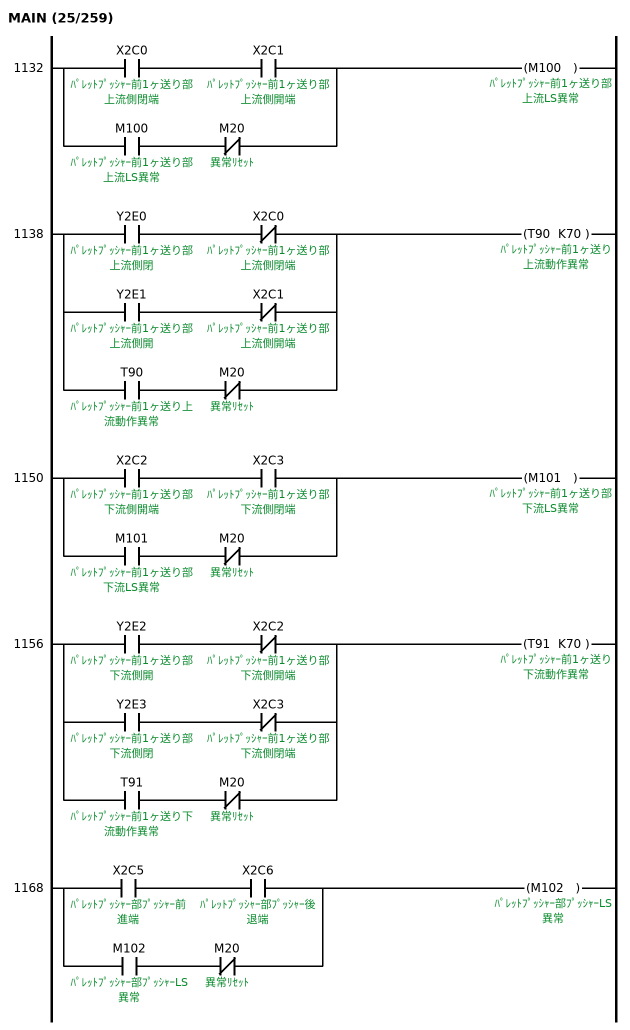
[picture p24: ladder of MAIN, rungs at steps 1132 to 1168]
1132  LD      X2C0  ; ﾊﾟﾚｯﾄﾌﾟｯｼｬｰ前1ヶ送り部上流側閉端
      AND     X2C1  ; ﾊﾟﾚｯﾄﾌﾟｯｼｬｰ前1ヶ送り部上流側開端
      LD      M100  ; ﾊﾟﾚｯﾄﾌﾟｯｼｬｰ前1ヶ送り部上流LS異常
      ANI     M20  ; 異常ﾘｾｯﾄ
      ORB
      OUT     M100  ; ﾊﾟﾚｯﾄﾌﾟｯｼｬｰ前1ヶ送り部上流LS異常
1138  LD      Y2E0  ; ﾊﾟﾚｯﾄﾌﾟｯｼｬｰ前1ヶ送り部上流側閉
      ANI     X2C0  ; ﾊﾟﾚｯﾄﾌﾟｯｼｬｰ前1ヶ送り部上流側閉端
      LD      Y2E1  ; ﾊﾟﾚｯﾄﾌﾟｯｼｬｰ前1ヶ送り部上流側開
      ANI     X2C1  ; ﾊﾟﾚｯﾄﾌﾟｯｼｬｰ前1ヶ送り部上流側開端
      ORB
      LD      T90  ; ﾊﾟﾚｯﾄﾌﾟｯｼｬｰ前1ヶ送り上流動作異常
      ANI     M20  ; 異常ﾘｾｯﾄ
      ORB
      OUT     T90 K70  ; ﾊﾟﾚｯﾄﾌﾟｯｼｬｰ前1ヶ送り上流動作異常
1150  LD      X2C2  ; ﾊﾟﾚｯﾄﾌﾟｯｼｬｰ前1ヶ送り部下流側開端
      AND     X2C3  ; ﾊﾟﾚｯﾄﾌﾟｯｼｬｰ前1ヶ送り部下流側閉端
      LD      M101  ; ﾊﾟﾚｯﾄﾌﾟｯｼｬｰ前1ヶ送り部下流LS異常
      ANI     M20  ; 異常ﾘｾｯﾄ
      ORB
      OUT     M101  ; ﾊﾟﾚｯﾄﾌﾟｯｼｬｰ前1ヶ送り部下流LS異常
1156  LD      Y2E2  ; ﾊﾟﾚｯﾄﾌﾟｯｼｬｰ前1ヶ送り部下流側開
      ANI     X2C2  ; ﾊﾟﾚｯﾄﾌﾟｯｼｬｰ前1ヶ送り部下流側開端
      LD      Y2E3  ; ﾊﾟﾚｯﾄﾌﾟｯｼｬｰ前1ヶ送り部下流側閉
      ANI     X2C3  ; ﾊﾟﾚｯﾄﾌﾟｯｼｬｰ前1ヶ送り部下流側閉端
      ORB
      LD      T91  ; ﾊﾟﾚｯﾄﾌﾟｯｼｬｰ前1ヶ送り下流動作異常
      ANI     M20  ; 異常ﾘｾｯﾄ
      ORB
      OUT     T91 K70  ; ﾊﾟﾚｯﾄﾌﾟｯｼｬｰ前1ヶ送り下流動作異常
1168  LD      X2C5  ; ﾊﾟﾚｯﾄﾌﾟｯｼｬｰ部ﾌﾟｯｼｬｰ前進端
      AND     X2C6  ; ﾊﾟﾚｯﾄﾌﾟｯｼｬｰ部ﾌﾟｯｼｬｰ後退端
      LD      M102  ; ﾊﾟﾚｯﾄﾌﾟｯｼｬｰ部ﾌﾟｯｼｬｰLS異常
      ANI     M20  ; 異常ﾘｾｯﾄ
      ORB
      OUT     M102  ; ﾊﾟﾚｯﾄﾌﾟｯｼｬｰ部ﾌﾟｯｼｬｰLS異常
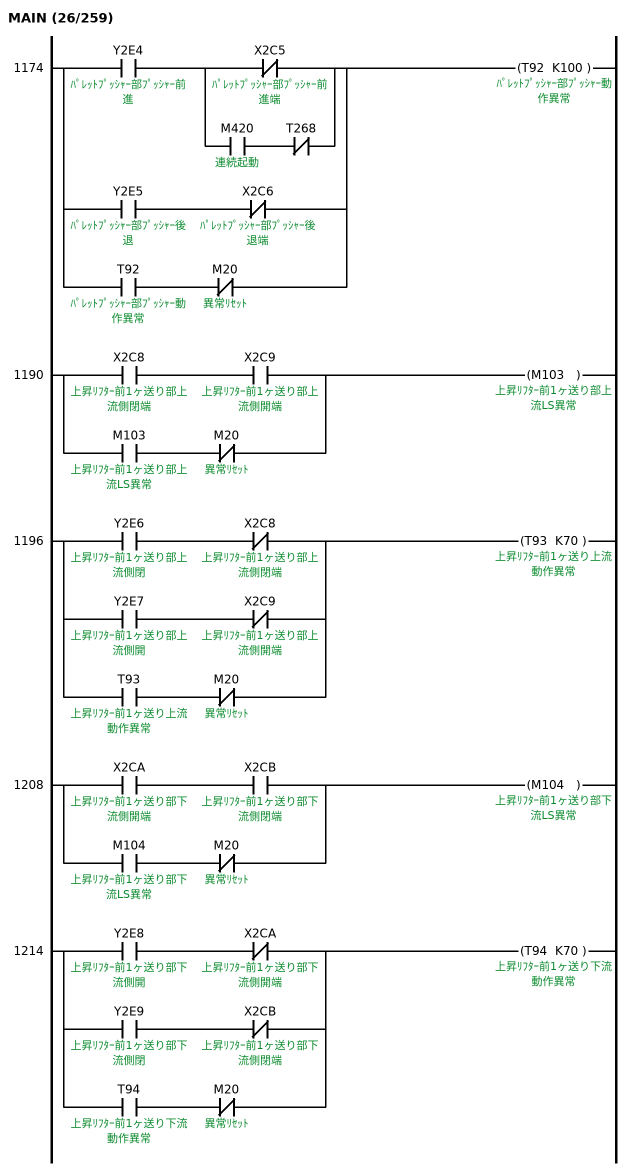
1174  LD      Y2E4  ; ﾊﾟﾚｯﾄﾌﾟｯｼｬｰ部ﾌﾟｯｼｬｰ前進
      LDI     X2C5  ; ﾊﾟﾚｯﾄﾌﾟｯｼｬｰ部ﾌﾟｯｼｬｰ前進端
      LD      M420  ; 連続起動
      ANI     T268
      ORB
      ANB
      LD      Y2E5  ; ﾊﾟﾚｯﾄﾌﾟｯｼｬｰ部ﾌﾟｯｼｬｰ後退
      ANI     X2C6  ; ﾊﾟﾚｯﾄﾌﾟｯｼｬｰ部ﾌﾟｯｼｬｰ後退端
      ORB
      LD      T92  ; ﾊﾟﾚｯﾄﾌﾟｯｼｬｰ部ﾌﾟｯｼｬｰ動作異常
      ANI     M20  ; 異常ﾘｾｯﾄ
      ORB
      OUT     T92 K100  ; ﾊﾟﾚｯﾄﾌﾟｯｼｬｰ部ﾌﾟｯｼｬｰ動作異常
1190  LD      X2C8  ; 上昇ﾘﾌﾀｰ前1ヶ送り部上流側閉端
      AND     X2C9  ; 上昇ﾘﾌﾀｰ前1ヶ送り部上流側開端
      LD      M103  ; 上昇ﾘﾌﾀｰ前1ヶ送り部上流LS異常
      ANI     M20  ; 異常ﾘｾｯﾄ
      ORB
      OUT     M103  ; 上昇ﾘﾌﾀｰ前1ヶ送り部上流LS異常
1196  LD      Y2E6  ; 上昇ﾘﾌﾀｰ前1ヶ送り部上流側閉
      ANI     X2C8  ; 上昇ﾘﾌﾀｰ前1ヶ送り部上流側閉端
      LD      Y2E7  ; 上昇ﾘﾌﾀｰ前1ヶ送り部上流側開
      ANI     X2C9  ; 上昇ﾘﾌﾀｰ前1ヶ送り部上流側開端
      ORB
      LD      T93  ; 上昇ﾘﾌﾀｰ前1ヶ送り上流動作異常
      ANI     M20  ; 異常ﾘｾｯﾄ
      ORB
      OUT     T93 K70  ; 上昇ﾘﾌﾀｰ前1ヶ送り上流動作異常
1208  LD      X2CA  ; 上昇ﾘﾌﾀｰ前1ヶ送り部下流側開端
      AND     X2CB  ; 上昇ﾘﾌﾀｰ前1ヶ送り部下流側閉端
      LD      M104  ; 上昇ﾘﾌﾀｰ前1ヶ送り部下流LS異常
      ANI     M20  ; 異常ﾘｾｯﾄ
      ORB
      OUT     M104  ; 上昇ﾘﾌﾀｰ前1ヶ送り部下流LS異常
1214  LD      Y2E8  ; 上昇ﾘﾌﾀｰ前1ヶ送り部下流側開
      ANI     X2CA  ; 上昇ﾘﾌﾀｰ前1ヶ送り部下流側開端
      LD      Y2E9  ; 上昇ﾘﾌﾀｰ前1ヶ送り部下流側閉
      ANI     X2CB  ; 上昇ﾘﾌﾀｰ前1ヶ送り部下流側閉端
      ORB
      LD      T94  ; 上昇ﾘﾌﾀｰ前1ヶ送り下流動作異常
      ANI     M20  ; 異常ﾘｾｯﾄ
      ORB
      OUT     T94 K70  ; 上昇ﾘﾌﾀｰ前1ヶ送り下流動作異常
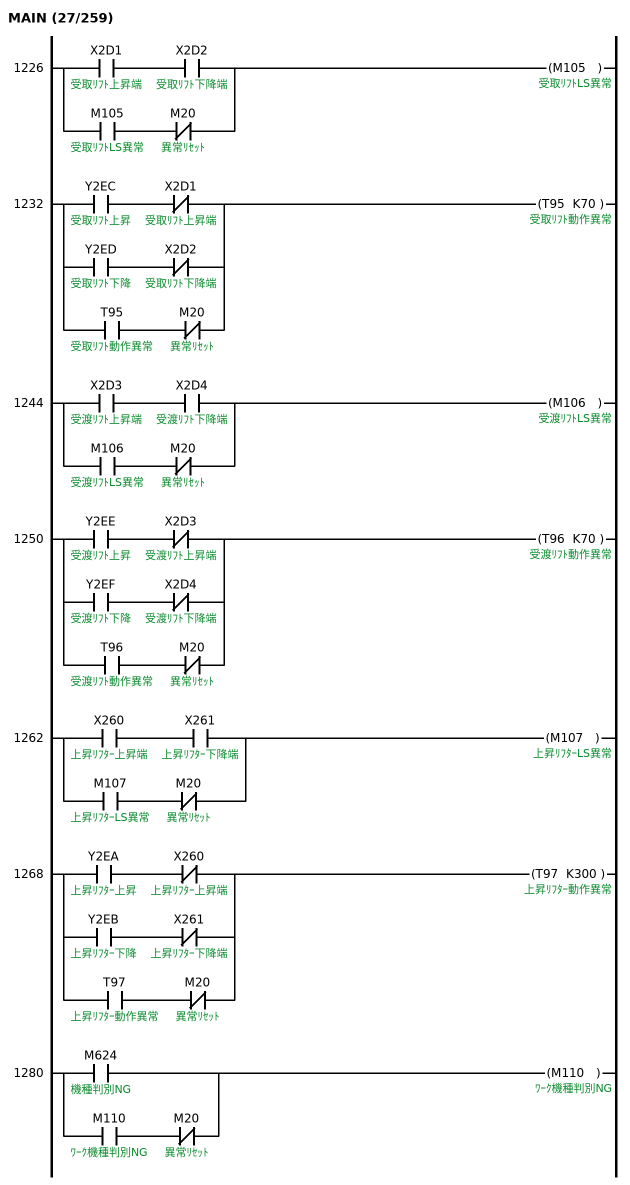
1226  LD      X2D1  ; 受取ﾘﾌﾄ上昇端
      AND     X2D2  ; 受取ﾘﾌﾄ下降端
      LD      M105  ; 受取ﾘﾌﾄLS異常
      ANI     M20  ; 異常ﾘｾｯﾄ
      ORB
      OUT     M105  ; 受取ﾘﾌﾄLS異常
1232  LD      Y2EC  ; 受取ﾘﾌﾄ上昇
      ANI     X2D1  ; 受取ﾘﾌﾄ上昇端
      LD      Y2ED  ; 受取ﾘﾌﾄ下降
      ANI     X2D2  ; 受取ﾘﾌﾄ下降端
      ORB
      LD      T95  ; 受取ﾘﾌﾄ動作異常
      ANI     M20  ; 異常ﾘｾｯﾄ
      ORB
      OUT     T95 K70  ; 受取ﾘﾌﾄ動作異常
1244  LD      X2D3  ; 受渡ﾘﾌﾄ上昇端
      AND     X2D4  ; 受渡ﾘﾌﾄ下降端
      LD      M106  ; 受渡ﾘﾌﾄLS異常
      ANI     M20  ; 異常ﾘｾｯﾄ
      ORB
      OUT     M106  ; 受渡ﾘﾌﾄLS異常
1250  LD      Y2EE  ; 受渡ﾘﾌﾄ上昇
      ANI     X2D3  ; 受渡ﾘﾌﾄ上昇端
      LD      Y2EF  ; 受渡ﾘﾌﾄ下降
      ANI     X2D4  ; 受渡ﾘﾌﾄ下降端
      ORB
      LD      T96  ; 受渡ﾘﾌﾄ動作異常
      ANI     M20  ; 異常ﾘｾｯﾄ
      ORB
      OUT     T96 K70  ; 受渡ﾘﾌﾄ動作異常
1262  LD      X260  ; 上昇ﾘﾌﾀｰ上昇端
      AND     X261  ; 上昇ﾘﾌﾀｰ下降端
      LD      M107  ; 上昇ﾘﾌﾀｰLS異常
      ANI     M20  ; 異常ﾘｾｯﾄ
      ORB
      OUT     M107  ; 上昇ﾘﾌﾀｰLS異常
1268  LD      Y2EA  ; 上昇ﾘﾌﾀｰ上昇
      ANI     X260  ; 上昇ﾘﾌﾀｰ上昇端
      LD      Y2EB  ; 上昇ﾘﾌﾀｰ下降
      ANI     X261  ; 上昇ﾘﾌﾀｰ下降端
      ORB
      LD      T97  ; 上昇ﾘﾌﾀｰ動作異常
      ANI     M20  ; 異常ﾘｾｯﾄ
      ORB
      OUT     T97 K300  ; 上昇ﾘﾌﾀｰ動作異常
1280  LD      M624  ; 機種判別NG
      LD      M110  ; ﾜｰｸ機種判別NG
      ANI     M20  ; 異常ﾘｾｯﾄ
      ORB
      OUT     M110  ; ﾜｰｸ機種判別NG
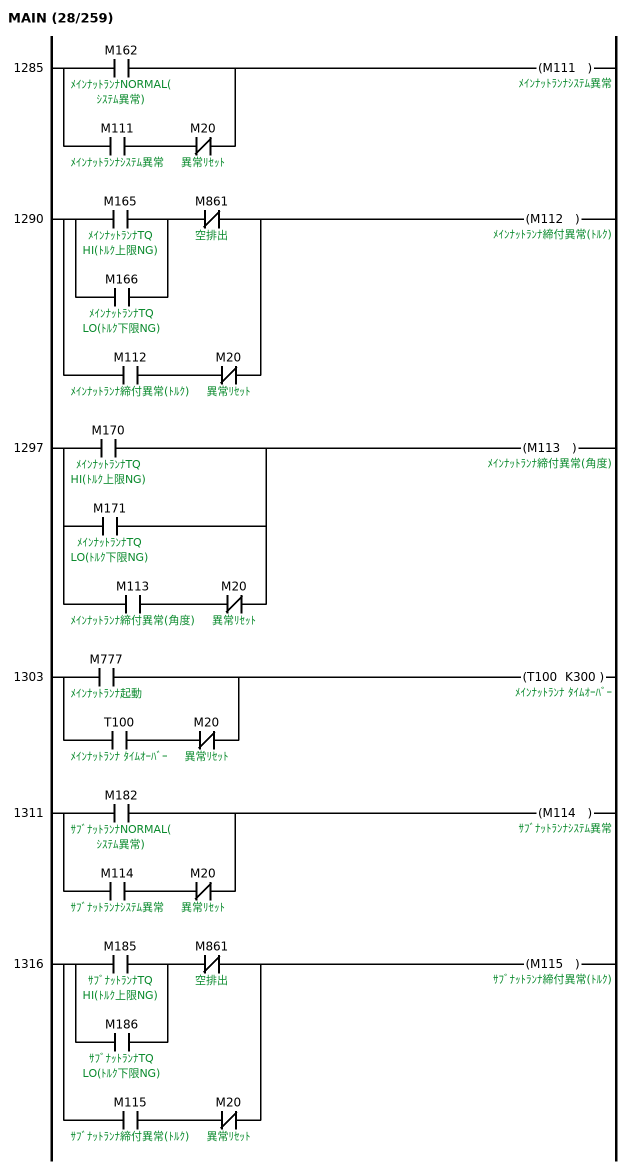
1285  LD      M162  ; ﾒｲﾝﾅｯﾄﾗﾝﾅNORMAL(ｼｽﾃﾑ異常)
      LD      M111  ; ﾒｲﾝﾅｯﾄﾗﾝﾅｼｽﾃﾑ異常
      ANI     M20  ; 異常ﾘｾｯﾄ
      ORB
      OUT     M111  ; ﾒｲﾝﾅｯﾄﾗﾝﾅｼｽﾃﾑ異常
1290  LD      M165  ; ﾒｲﾝﾅｯﾄﾗﾝﾅTQ HI(ﾄﾙｸ上限NG)
      OR      M166  ; ﾒｲﾝﾅｯﾄﾗﾝﾅTQ LO(ﾄﾙｸ下限NG)
      ANI     M861  ; 空排出
      LD      M112  ; ﾒｲﾝﾅｯﾄﾗﾝﾅ締付異常(ﾄﾙｸ)
      ANI     M20  ; 異常ﾘｾｯﾄ
      ORB
      OUT     M112  ; ﾒｲﾝﾅｯﾄﾗﾝﾅ締付異常(ﾄﾙｸ)
1297  LD      M170  ; ﾒｲﾝﾅｯﾄﾗﾝﾅTQ HI(ﾄﾙｸ上限NG)
      OR      M171  ; ﾒｲﾝﾅｯﾄﾗﾝﾅTQ LO(ﾄﾙｸ下限NG)
      LD      M113  ; ﾒｲﾝﾅｯﾄﾗﾝﾅ締付異常(角度)
      ANI     M20  ; 異常ﾘｾｯﾄ
      ORB
      OUT     M113  ; ﾒｲﾝﾅｯﾄﾗﾝﾅ締付異常(角度)
1303  LD      M777  ; ﾒｲﾝﾅｯﾄﾗﾝﾅ起動
      LD      T100  ; ﾒｲﾝﾅｯﾄﾗﾝﾅ ﾀｲﾑｵｰﾊﾞｰ
      ANI     M20  ; 異常ﾘｾｯﾄ
      ORB
      OUT     T100 K300  ; ﾒｲﾝﾅｯﾄﾗﾝﾅ ﾀｲﾑｵｰﾊﾞｰ
1311  LD      M182  ; ｻﾌﾞﾅｯﾄﾗﾝﾅNORMAL(ｼｽﾃﾑ異常)
      LD      M114  ; ｻﾌﾞﾅｯﾄﾗﾝﾅｼｽﾃﾑ異常
      ANI     M20  ; 異常ﾘｾｯﾄ
      ORB
      OUT     M114  ; ｻﾌﾞﾅｯﾄﾗﾝﾅｼｽﾃﾑ異常
1316  LD      M185  ; ｻﾌﾞﾅｯﾄﾗﾝﾅTQ HI(ﾄﾙｸ上限NG)
      OR      M186  ; ｻﾌﾞﾅｯﾄﾗﾝﾅTQ LO(ﾄﾙｸ下限NG)
      ANI     M861  ; 空排出
      LD      M115  ; ｻﾌﾞﾅｯﾄﾗﾝﾅ締付異常(ﾄﾙｸ)
      ANI     M20  ; 異常ﾘｾｯﾄ
      ORB
      OUT     M115  ; ｻﾌﾞﾅｯﾄﾗﾝﾅ締付異常(ﾄﾙｸ)
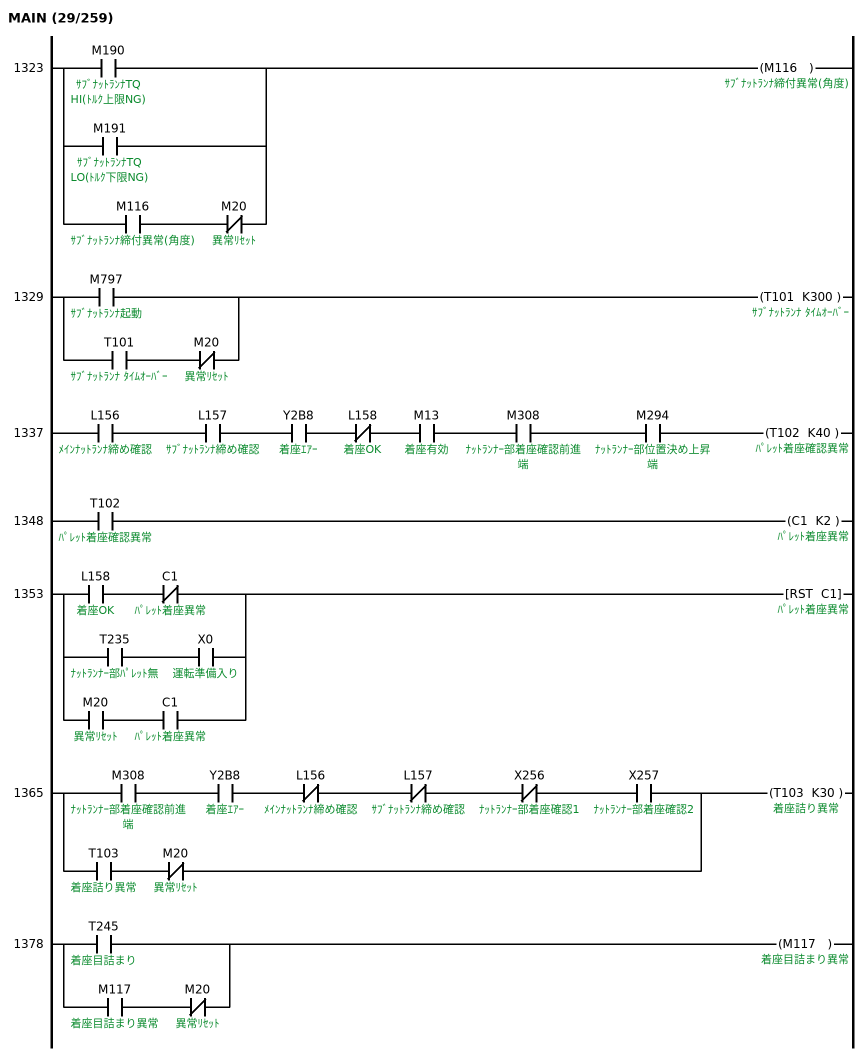
1323  LD      M190  ; ｻﾌﾞﾅｯﾄﾗﾝﾅTQ HI(ﾄﾙｸ上限NG)
      OR      M191  ; ｻﾌﾞﾅｯﾄﾗﾝﾅTQ LO(ﾄﾙｸ下限NG)
      LD      M116  ; ｻﾌﾞﾅｯﾄﾗﾝﾅ締付異常(角度)
      ANI     M20  ; 異常ﾘｾｯﾄ
      ORB
      OUT     M116  ; ｻﾌﾞﾅｯﾄﾗﾝﾅ締付異常(角度)
1329  LD      M797  ; ｻﾌﾞﾅｯﾄﾗﾝﾅ起動
      LD      T101  ; ｻﾌﾞﾅｯﾄﾗﾝﾅ ﾀｲﾑｵｰﾊﾞｰ
      ANI     M20  ; 異常ﾘｾｯﾄ
      ORB
      OUT     T101 K300  ; ｻﾌﾞﾅｯﾄﾗﾝﾅ ﾀｲﾑｵｰﾊﾞｰ
1337  LD      L156  ; ﾒｲﾝﾅｯﾄﾗﾝﾅ締め確認
      AND     L157  ; ｻﾌﾞﾅｯﾄﾗﾝﾅ締め確認
      AND     Y2B8  ; 着座ｴｱｰ
      ANI     L158  ; 着座OK
      AND     M13  ; 着座有効
      AND     M308  ; ﾅｯﾄﾗﾝﾅｰ部着座確認前進端
      AND     M294  ; ﾅｯﾄﾗﾝﾅｰ部位置決め上昇端
      OUT     T102 K40  ; ﾊﾟﾚｯﾄ着座確認異常
1348  LD      T102  ; ﾊﾟﾚｯﾄ着座確認異常
      OUT     C1 K2  ; ﾊﾟﾚｯﾄ着座異常
1353  LD      L158  ; 着座OK
      ANI     C1  ; ﾊﾟﾚｯﾄ着座異常
      LD      T235  ; ﾅｯﾄﾗﾝﾅｰ部ﾊﾟﾚｯﾄ無
      AND     X0  ; 運転準備入り
      ORB
      LD      M20  ; 異常ﾘｾｯﾄ
      AND     C1  ; ﾊﾟﾚｯﾄ着座異常
      ORB
      RST     C1  ; ﾊﾟﾚｯﾄ着座異常
1365  LD      M308  ; ﾅｯﾄﾗﾝﾅｰ部着座確認前進端
      AND     Y2B8  ; 着座ｴｱｰ
      ANI     L156  ; ﾒｲﾝﾅｯﾄﾗﾝﾅ締め確認
      ANI     L157  ; ｻﾌﾞﾅｯﾄﾗﾝﾅ締め確認
      ANI     X256  ; ﾅｯﾄﾗﾝﾅｰ部着座確認1
      AND     X257  ; ﾅｯﾄﾗﾝﾅｰ部着座確認2
      LD      T103  ; 着座詰り異常
      ANI     M20  ; 異常ﾘｾｯﾄ
      ORB
      OUT     T103 K30  ; 着座詰り異常
1378  LD      T245  ; 着座目詰まり
      LD      M117  ; 着座目詰まり異常
      ANI     M20  ; 異常ﾘｾｯﾄ
      ORB
      OUT     M117  ; 着座目詰まり異常
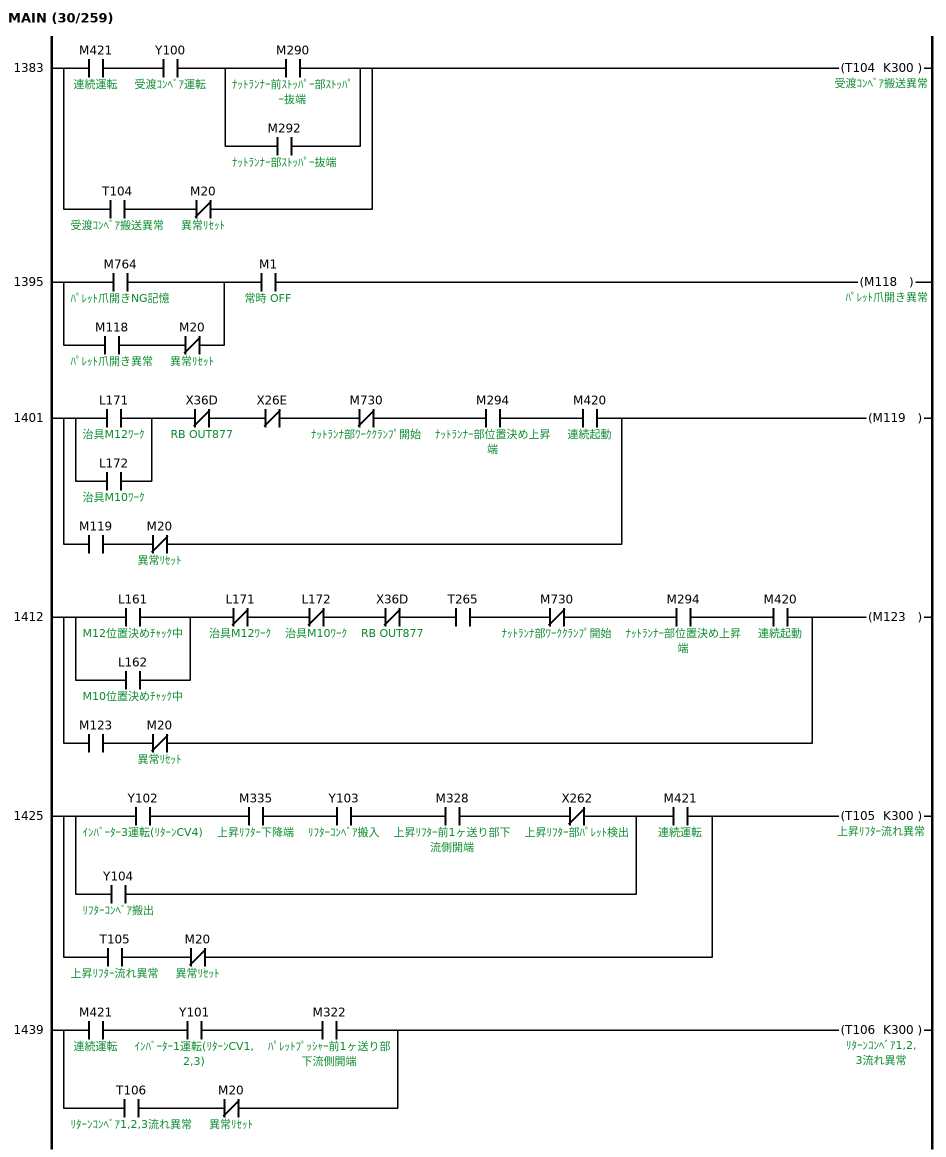
1383  LD      M421  ; 連続運転
      AND     Y100  ; 受渡ｺﾝﾍﾞｱ運転
      LD      M290  ; ﾅｯﾄﾗﾝﾅｰ前ｽﾄｯﾊﾟｰ部ｽﾄｯﾊﾟｰ抜端
      OR      M292  ; ﾅｯﾄﾗﾝﾅｰ部ｽﾄｯﾊﾟｰ抜端
      ANB
      LD      T104  ; 受渡ｺﾝﾍﾞｱ搬送異常
      ANI     M20  ; 異常ﾘｾｯﾄ
      ORB
      OUT     T104 K300  ; 受渡ｺﾝﾍﾞｱ搬送異常
1395  LD      M764  ; ﾊﾟﾚｯﾄ爪開きNG記憶
      LD      M118  ; ﾊﾟﾚｯﾄ爪開き異常
      ANI     M20  ; 異常ﾘｾｯﾄ
      ORB
      AND     M1  ; 常時 OFF
      OUT     M118  ; ﾊﾟﾚｯﾄ爪開き異常
1401  LD      L171  ; 治具M12ﾜｰｸ
      OR      L172  ; 治具M10ﾜｰｸ
      ANI     X36D  ; RB OUT877
      ANI     X26E
      ANI     M730  ; ﾅｯﾄﾗﾝﾅ部ﾜｰｸｸﾗﾝﾌﾟ開始
      AND     M294  ; ﾅｯﾄﾗﾝﾅｰ部位置決め上昇端
      AND     M420  ; 連続起動
      LD      M119
      ANI     M20  ; 異常ﾘｾｯﾄ
      ORB
      OUT     M119
1412  LD      L161  ; M12位置決めﾁｬｯｸ中
      OR      L162  ; M10位置決めﾁｬｯｸ中
      ANI     L171  ; 治具M12ﾜｰｸ
      ANI     L172  ; 治具M10ﾜｰｸ
      ANI     X36D  ; RB OUT877
      AND     T265
      ANI     M730  ; ﾅｯﾄﾗﾝﾅ部ﾜｰｸｸﾗﾝﾌﾟ開始
      AND     M294  ; ﾅｯﾄﾗﾝﾅｰ部位置決め上昇端
      AND     M420  ; 連続起動
      LD      M123
      ANI     M20  ; 異常ﾘｾｯﾄ
      ORB
      OUT     M123
1425  LD      Y102  ; ｲﾝﾊﾞｰﾀｰ3運転(ﾘﾀｰﾝCV4)
      AND     M335  ; 上昇ﾘﾌﾀｰ下降端
      AND     Y103  ; ﾘﾌﾀｰｺﾝﾍﾞｱ搬入
      AND     M328  ; 上昇ﾘﾌﾀｰ前1ヶ送り部下流側開端
      ANI     X262  ; 上昇ﾘﾌﾀｰ部ﾊﾟﾚｯﾄ検出
      OR      Y104  ; ﾘﾌﾀｰｺﾝﾍﾞｱ搬出
      AND     M421  ; 連続運転
      LD      T105  ; 上昇ﾘﾌﾀｰ流れ異常
      ANI     M20  ; 異常ﾘｾｯﾄ
      ORB
      OUT     T105 K300  ; 上昇ﾘﾌﾀｰ流れ異常
1439  LD      M421  ; 連続運転
      AND     Y101  ; ｲﾝﾊﾞｰﾀｰ1運転(ﾘﾀｰﾝCV1,2,3)
      AND     M322  ; ﾊﾟﾚｯﾄﾌﾟｯｼｬｰ前1ヶ送り部下流側開端
      LD      T106  ; ﾘﾀｰﾝｺﾝﾍﾞｱ1,2,3流れ異常
      ANI     M20  ; 異常ﾘｾｯﾄ
      ORB
      OUT     T106 K300  ; ﾘﾀｰﾝｺﾝﾍﾞｱ1,2,3流れ異常
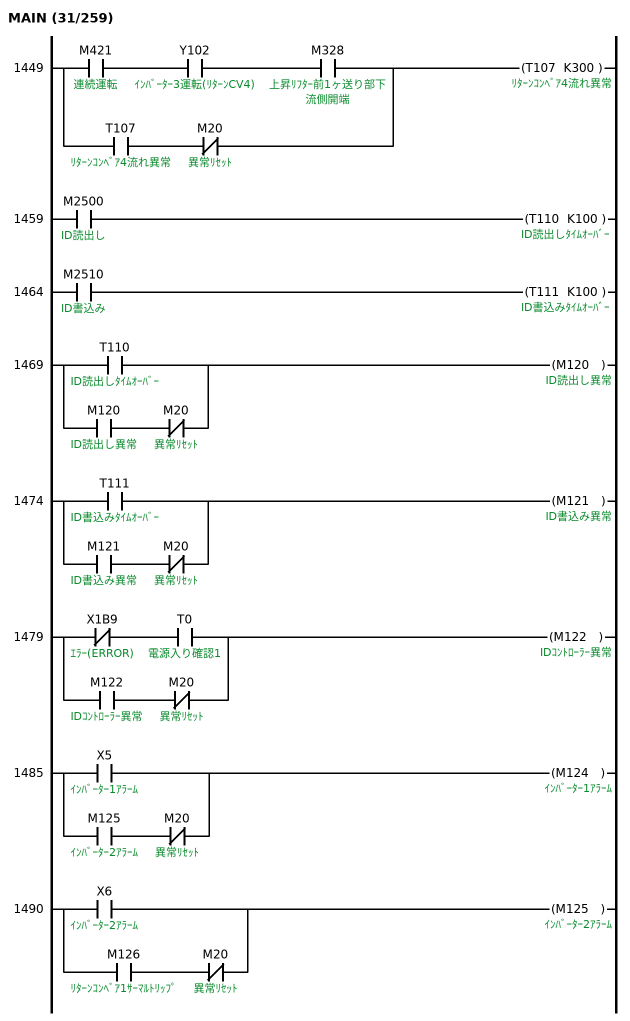
1449  LD      M421  ; 連続運転
      AND     Y102  ; ｲﾝﾊﾞｰﾀｰ3運転(ﾘﾀｰﾝCV4)
      AND     M328  ; 上昇ﾘﾌﾀｰ前1ヶ送り部下流側開端
      LD      T107  ; ﾘﾀｰﾝｺﾝﾍﾞｱ4流れ異常
      ANI     M20  ; 異常ﾘｾｯﾄ
      ORB
      OUT     T107 K300  ; ﾘﾀｰﾝｺﾝﾍﾞｱ4流れ異常
1459  LD      M2500  ; ID読出し
      OUT     T110 K100  ; ID読出しﾀｲﾑｵｰﾊﾞｰ
1464  LD      M2510  ; ID書込み
      OUT     T111 K100  ; ID書込みﾀｲﾑｵｰﾊﾞｰ
1469  LD      T110  ; ID読出しﾀｲﾑｵｰﾊﾞｰ
      LD      M120  ; ID読出し異常
      ANI     M20  ; 異常ﾘｾｯﾄ
      ORB
      OUT     M120  ; ID読出し異常
1474  LD      T111  ; ID書込みﾀｲﾑｵｰﾊﾞｰ
      LD      M121  ; ID書込み異常
      ANI     M20  ; 異常ﾘｾｯﾄ
      ORB
      OUT     M121  ; ID書込み異常
1479  LDI     X1B9  ; ｴﾗｰ(ERROR)
      AND     T0  ; 電源入り確認1
      LD      M122  ; IDｺﾝﾄﾛｰﾗｰ異常
      ANI     M20  ; 異常ﾘｾｯﾄ
      ORB
      OUT     M122  ; IDｺﾝﾄﾛｰﾗｰ異常
1485  LD      X5  ; ｲﾝﾊﾞｰﾀｰ1ｱﾗｰﾑ
      LD      M125  ; ｲﾝﾊﾞｰﾀｰ2ｱﾗｰﾑ
      ANI     M20  ; 異常ﾘｾｯﾄ
      ORB
      OUT     M124  ; ｲﾝﾊﾞｰﾀｰ1ｱﾗｰﾑ
1490  LD      X6  ; ｲﾝﾊﾞｰﾀｰ2ｱﾗｰﾑ
      LD      M126  ; ﾘﾀｰﾝｺﾝﾍﾞｱ1ｻｰﾏﾙﾄﾘｯﾌﾟ
      ANI     M20  ; 異常ﾘｾｯﾄ
      ORB
      OUT     M125  ; ｲﾝﾊﾞｰﾀｰ2ｱﾗｰﾑ
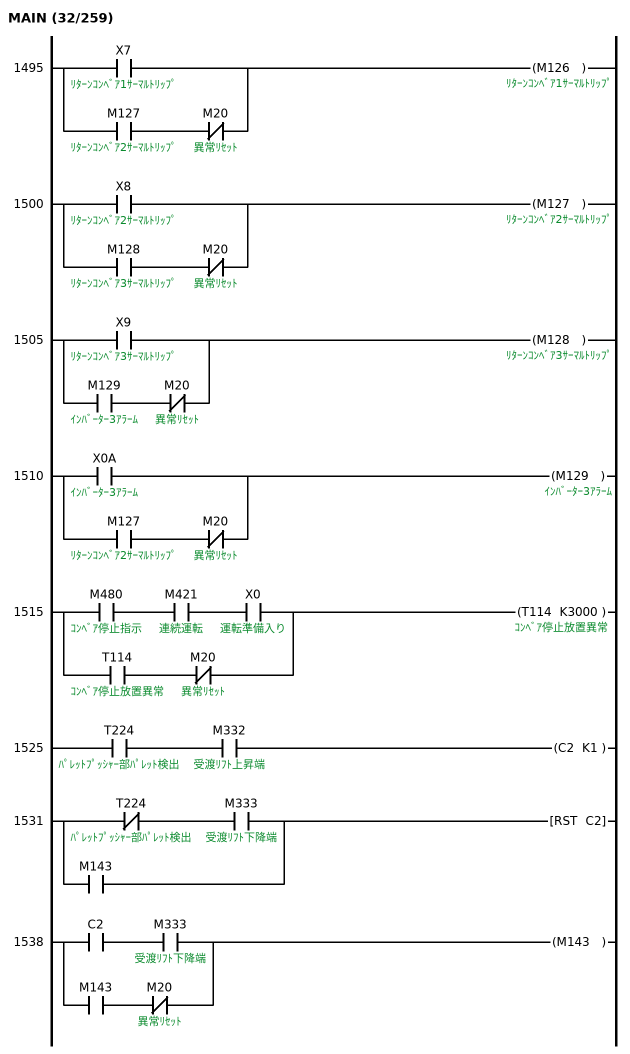
1495  LD      X7  ; ﾘﾀｰﾝｺﾝﾍﾞｱ1ｻｰﾏﾙﾄﾘｯﾌﾟ
      LD      M127  ; ﾘﾀｰﾝｺﾝﾍﾞｱ2ｻｰﾏﾙﾄﾘｯﾌﾟ
      ANI     M20  ; 異常ﾘｾｯﾄ
      ORB
      OUT     M126  ; ﾘﾀｰﾝｺﾝﾍﾞｱ1ｻｰﾏﾙﾄﾘｯﾌﾟ
1500  LD      X8  ; ﾘﾀｰﾝｺﾝﾍﾞｱ2ｻｰﾏﾙﾄﾘｯﾌﾟ
      LD      M128  ; ﾘﾀｰﾝｺﾝﾍﾞｱ3ｻｰﾏﾙﾄﾘｯﾌﾟ
      ANI     M20  ; 異常ﾘｾｯﾄ
      ORB
      OUT     M127  ; ﾘﾀｰﾝｺﾝﾍﾞｱ2ｻｰﾏﾙﾄﾘｯﾌﾟ
1505  LD      X9  ; ﾘﾀｰﾝｺﾝﾍﾞｱ3ｻｰﾏﾙﾄﾘｯﾌﾟ
      LD      M129  ; ｲﾝﾊﾞｰﾀｰ3ｱﾗｰﾑ
      ANI     M20  ; 異常ﾘｾｯﾄ
      ORB
      OUT     M128  ; ﾘﾀｰﾝｺﾝﾍﾞｱ3ｻｰﾏﾙﾄﾘｯﾌﾟ
1510  LD      X0A  ; ｲﾝﾊﾞｰﾀｰ3ｱﾗｰﾑ
      LD      M127  ; ﾘﾀｰﾝｺﾝﾍﾞｱ2ｻｰﾏﾙﾄﾘｯﾌﾟ
      ANI     M20  ; 異常ﾘｾｯﾄ
      ORB
      OUT     M129  ; ｲﾝﾊﾞｰﾀｰ3ｱﾗｰﾑ
1515  LD      M480  ; ｺﾝﾍﾞｱ停止指示
      AND     M421  ; 連続運転
      AND     X0  ; 運転準備入り
      LD      T114  ; ｺﾝﾍﾞｱ停止放置異常
      ANI     M20  ; 異常ﾘｾｯﾄ
      ORB
      OUT     T114 K3000  ; ｺﾝﾍﾞｱ停止放置異常
1525  LD      T224  ; ﾊﾟﾚｯﾄﾌﾟｯｼｬｰ部ﾊﾟﾚｯﾄ検出
      AND     M332  ; 受渡ﾘﾌﾄ上昇端
      OUT     C2 K1
1531  LDI     T224  ; ﾊﾟﾚｯﾄﾌﾟｯｼｬｰ部ﾊﾟﾚｯﾄ検出
      AND     M333  ; 受渡ﾘﾌﾄ下降端
      OR      M143
      RST     C2
1538  LD      C2
      AND     M333  ; 受渡ﾘﾌﾄ下降端
      LD      M143
      ANI     M20  ; 異常ﾘｾｯﾄ
      ORB
      OUT     M143
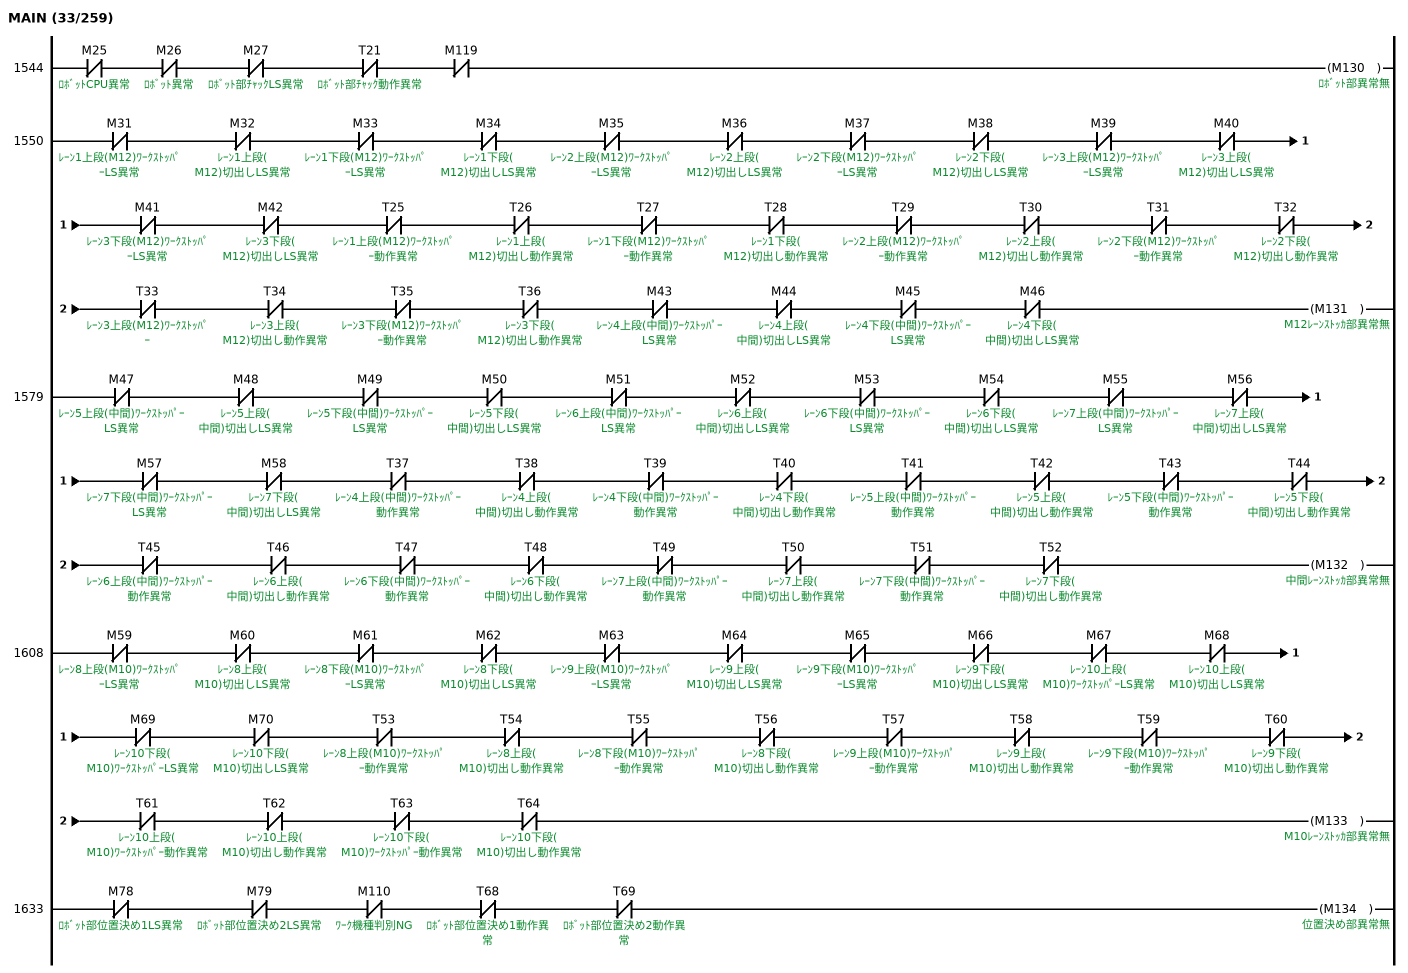
1544  LDI     M25  ; ﾛﾎﾞｯﾄCPU異常
      ANI     M26  ; ﾛﾎﾞｯﾄ異常
      ANI     M27  ; ﾛﾎﾞｯﾄ部ﾁｬｯｸLS異常
      ANI     T21  ; ﾛﾎﾞｯﾄ部ﾁｬｯｸ動作異常
      ANI     M119
      OUT     M130  ; ﾛﾎﾞｯﾄ部異常無
1550  LDI     M31  ; ﾚｰﾝ1上段(M12)ﾜｰｸｽﾄｯﾊﾟｰLS異常
      ANI     M32  ; ﾚｰﾝ1上段(M12)切出しLS異常
      ANI     M33  ; ﾚｰﾝ1下段(M12)ﾜｰｸｽﾄｯﾊﾟｰLS異常
      ANI     M34  ; ﾚｰﾝ1下段(M12)切出しLS異常
      ANI     M35  ; ﾚｰﾝ2上段(M12)ﾜｰｸｽﾄｯﾊﾟｰLS異常
      ANI     M36  ; ﾚｰﾝ2上段(M12)切出しLS異常
      ANI     M37  ; ﾚｰﾝ2下段(M12)ﾜｰｸｽﾄｯﾊﾟｰLS異常
      ANI     M38  ; ﾚｰﾝ2下段(M12)切出しLS異常
      ANI     M39  ; ﾚｰﾝ3上段(M12)ﾜｰｸｽﾄｯﾊﾟｰLS異常
      ANI     M40  ; ﾚｰﾝ3上段(M12)切出しLS異常
      ANI     M41  ; ﾚｰﾝ3下段(M12)ﾜｰｸｽﾄｯﾊﾟｰLS異常
      ANI     M42  ; ﾚｰﾝ3下段(M12)切出しLS異常
      ANI     T25  ; ﾚｰﾝ1上段(M12)ﾜｰｸｽﾄｯﾊﾟｰ動作異常
      ANI     T26  ; ﾚｰﾝ1上段(M12)切出し動作異常
      ANI     T27  ; ﾚｰﾝ1下段(M12)ﾜｰｸｽﾄｯﾊﾟｰ動作異常
      ANI     T28  ; ﾚｰﾝ1下段(M12)切出し動作異常
      ANI     T29  ; ﾚｰﾝ2上段(M12)ﾜｰｸｽﾄｯﾊﾟｰ動作異常
      ANI     T30  ; ﾚｰﾝ2上段(M12)切出し動作異常
      ANI     T31  ; ﾚｰﾝ2下段(M12)ﾜｰｸｽﾄｯﾊﾟｰ動作異常
      ANI     T32  ; ﾚｰﾝ2下段(M12)切出し動作異常
      ANI     T33  ; ﾚｰﾝ3上段(M12)ﾜｰｸｽﾄｯﾊﾟｰ
      ANI     T34  ; ﾚｰﾝ3上段(M12)切出し動作異常
      ANI     T35  ; ﾚｰﾝ3下段(M12)ﾜｰｸｽﾄｯﾊﾟｰ動作異常
      ANI     T36  ; ﾚｰﾝ3下段(M12)切出し動作異常
      ANI     M43  ; ﾚｰﾝ4上段(中間)ﾜｰｸｽﾄｯﾊﾟｰLS異常
      ANI     M44  ; ﾚｰﾝ4上段(中間)切出しLS異常
      ANI     M45  ; ﾚｰﾝ4下段(中間)ﾜｰｸｽﾄｯﾊﾟｰLS異常
      ANI     M46  ; ﾚｰﾝ4下段(中間)切出しLS異常
      OUT     M131  ; M12ﾚｰﾝｽﾄｯｶ部異常無
1579  LDI     M47  ; ﾚｰﾝ5上段(中間)ﾜｰｸｽﾄｯﾊﾟｰLS異常
      ANI     M48  ; ﾚｰﾝ5上段(中間)切出しLS異常
      ANI     M49  ; ﾚｰﾝ5下段(中間)ﾜｰｸｽﾄｯﾊﾟｰLS異常
      ANI     M50  ; ﾚｰﾝ5下段(中間)切出しLS異常
      ANI     M51  ; ﾚｰﾝ6上段(中間)ﾜｰｸｽﾄｯﾊﾟｰLS異常
      ANI     M52  ; ﾚｰﾝ6上段(中間)切出しLS異常
      ANI     M53  ; ﾚｰﾝ6下段(中間)ﾜｰｸｽﾄｯﾊﾟｰLS異常
      ANI     M54  ; ﾚｰﾝ6下段(中間)切出しLS異常
      ANI     M55  ; ﾚｰﾝ7上段(中間)ﾜｰｸｽﾄｯﾊﾟｰLS異常
      ANI     M56  ; ﾚｰﾝ7上段(中間)切出しLS異常
      ANI     M57  ; ﾚｰﾝ7下段(中間)ﾜｰｸｽﾄｯﾊﾟｰLS異常
      ANI     M58  ; ﾚｰﾝ7下段(中間)切出しLS異常
      ANI     T37  ; ﾚｰﾝ4上段(中間)ﾜｰｸｽﾄｯﾊﾟｰ動作異常
      ANI     T38  ; ﾚｰﾝ4上段(中間)切出し動作異常
      ANI     T39  ; ﾚｰﾝ4下段(中間)ﾜｰｸｽﾄｯﾊﾟｰ動作異常
      ANI     T40  ; ﾚｰﾝ4下段(中間)切出し動作異常
      ANI     T41  ; ﾚｰﾝ5上段(中間)ﾜｰｸｽﾄｯﾊﾟｰ動作異常
      ANI     T42  ; ﾚｰﾝ5上段(中間)切出し動作異常
      ANI     T43  ; ﾚｰﾝ5下段(中間)ﾜｰｸｽﾄｯﾊﾟｰ動作異常
      ANI     T44  ; ﾚｰﾝ5下段(中間)切出し動作異常
      ANI     T45  ; ﾚｰﾝ6上段(中間)ﾜｰｸｽﾄｯﾊﾟｰ動作異常
      ANI     T46  ; ﾚｰﾝ6上段(中間)切出し動作異常
      ANI     T47  ; ﾚｰﾝ6下段(中間)ﾜｰｸｽﾄｯﾊﾟｰ動作異常
      ANI     T48  ; ﾚｰﾝ6下段(中間)切出し動作異常
      ANI     T49  ; ﾚｰﾝ7上段(中間)ﾜｰｸｽﾄｯﾊﾟｰ動作異常
      ANI     T50  ; ﾚｰﾝ7上段(中間)切出し動作異常
      ANI     T51  ; ﾚｰﾝ7下段(中間)ﾜｰｸｽﾄｯﾊﾟｰ動作異常
      ANI     T52  ; ﾚｰﾝ7下段(中間)切出し動作異常
      OUT     M132  ; 中間ﾚｰﾝｽﾄｯｶ部異常無
1608  LDI     M59  ; ﾚｰﾝ8上段(M10)ﾜｰｸｽﾄｯﾊﾟｰLS異常
      ANI     M60  ; ﾚｰﾝ8上段(M10)切出しLS異常
      ANI     M61  ; ﾚｰﾝ8下段(M10)ﾜｰｸｽﾄｯﾊﾟｰLS異常
      ANI     M62  ; ﾚｰﾝ8下段(M10)切出しLS異常
      ANI     M63  ; ﾚｰﾝ9上段(M10)ﾜｰｸｽﾄｯﾊﾟｰLS異常
      ANI     M64  ; ﾚｰﾝ9上段(M10)切出しLS異常
      ANI     M65  ; ﾚｰﾝ9下段(M10)ﾜｰｸｽﾄｯﾊﾟｰLS異常
      ANI     M66  ; ﾚｰﾝ9下段(M10)切出しLS異常
      ANI     M67  ; ﾚｰﾝ10上段(M10)ﾜｰｸｽﾄｯﾊﾟｰLS異常
      ANI     M68  ; ﾚｰﾝ10上段(M10)切出しLS異常
      ANI     M69  ; ﾚｰﾝ10下段(M10)ﾜｰｸｽﾄｯﾊﾟｰLS異常
      ANI     M70  ; ﾚｰﾝ10下段(M10)切出しLS異常
      ANI     T53  ; ﾚｰﾝ8上段(M10)ﾜｰｸｽﾄｯﾊﾟｰ動作異常
      ANI     T54  ; ﾚｰﾝ8上段(M10)切出し動作異常
      ANI     T55  ; ﾚｰﾝ8下段(M10)ﾜｰｸｽﾄｯﾊﾟｰ動作異常
      ANI     T56  ; ﾚｰﾝ8下段(M10)切出し動作異常
      ANI     T57  ; ﾚｰﾝ9上段(M10)ﾜｰｸｽﾄｯﾊﾟｰ動作異常
      ANI     T58  ; ﾚｰﾝ9上段(M10)切出し動作異常
      ANI     T59  ; ﾚｰﾝ9下段(M10)ﾜｰｸｽﾄｯﾊﾟｰ動作異常
      ANI     T60  ; ﾚｰﾝ9下段(M10)切出し動作異常
      ANI     T61  ; ﾚｰﾝ10上段(M10)ﾜｰｸｽﾄｯﾊﾟｰ動作異常
      ANI     T62  ; ﾚｰﾝ10上段(M10)切出し動作異常
      ANI     T63  ; ﾚｰﾝ10下段(M10)ﾜｰｸｽﾄｯﾊﾟｰ動作異常
      ANI     T64  ; ﾚｰﾝ10下段(M10)切出し動作異常
      OUT     M133  ; M10ﾚｰﾝｽﾄｯｶ部異常無
1633  LDI     M78  ; ﾛﾎﾞｯﾄ部位置決め1LS異常
      ANI     M79  ; ﾛﾎﾞｯﾄ部位置決め2LS異常
      ANI     M110  ; ﾜｰｸ機種判別NG
      ANI     T68  ; ﾛﾎﾞｯﾄ部位置決め1動作異常
      ANI     T69  ; ﾛﾎﾞｯﾄ部位置決め2動作異常
      OUT     M134  ; 位置決め部異常無
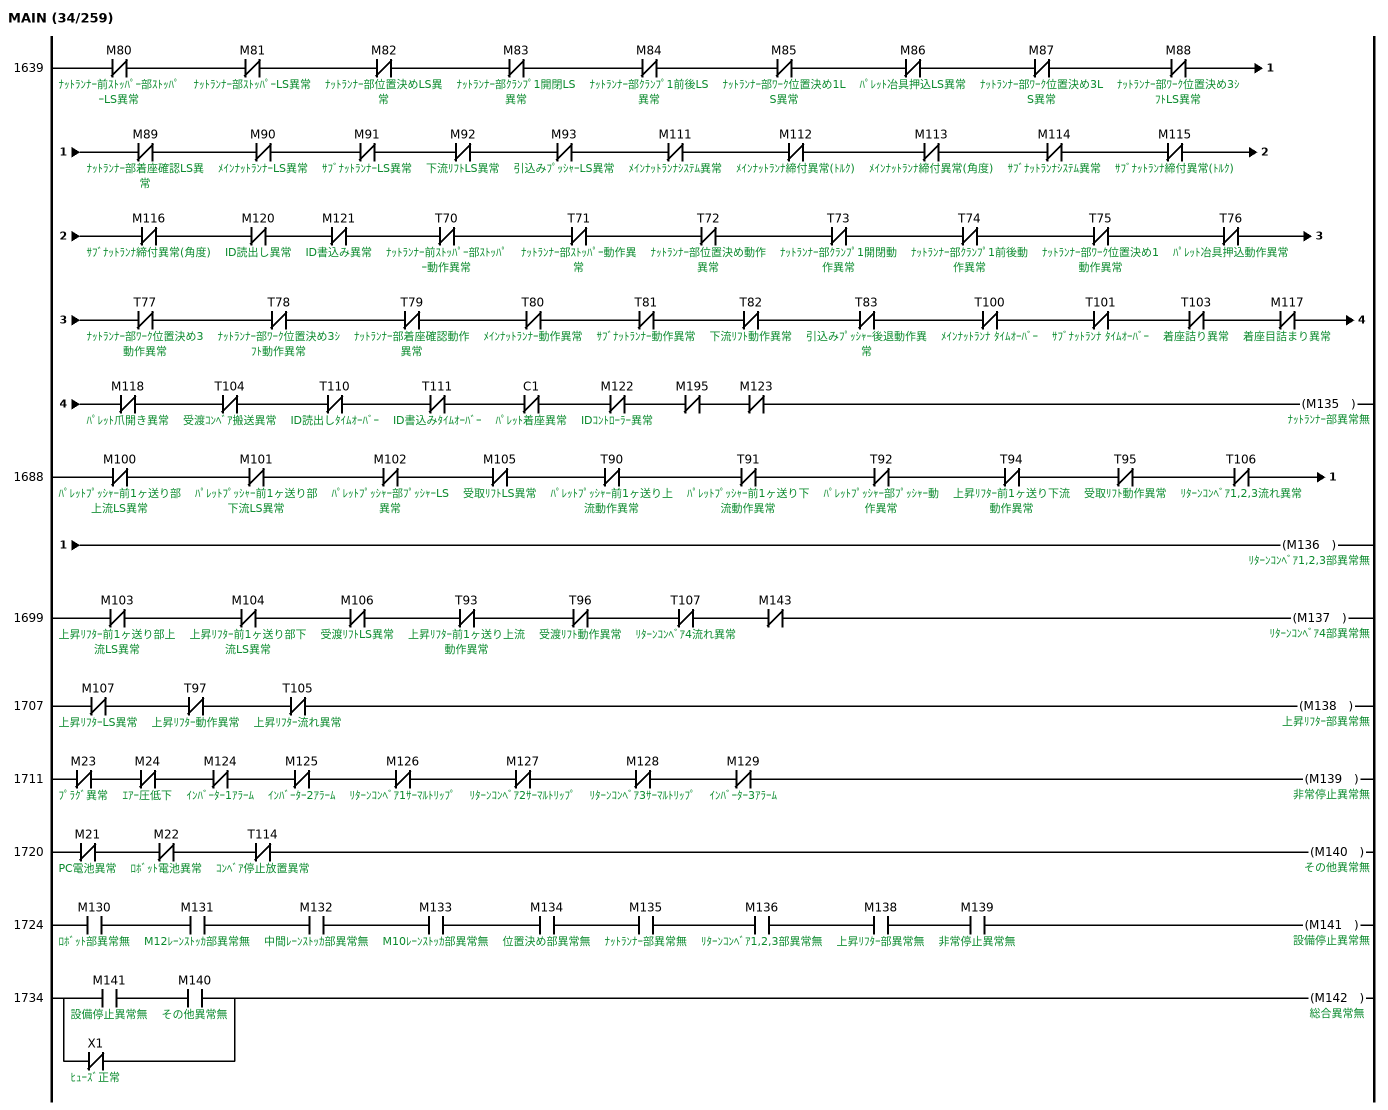
1639  LDI     M80  ; ﾅｯﾄﾗﾝﾅｰ前ｽﾄｯﾊﾟｰ部ｽﾄｯﾊﾟｰLS異常
      ANI     M81  ; ﾅｯﾄﾗﾝﾅｰ部ｽﾄｯﾊﾟｰLS異常
      ANI     M82  ; ﾅｯﾄﾗﾝﾅｰ部位置決めLS異常
      ANI     M83  ; ﾅｯﾄﾗﾝﾅｰ部ｸﾗﾝﾌﾟ1開閉LS異常
      ANI     M84  ; ﾅｯﾄﾗﾝﾅｰ部ｸﾗﾝﾌﾟ1前後LS異常
      ANI     M85  ; ﾅｯﾄﾗﾝﾅｰ部ﾜｰｸ位置決め1LS異常
      ANI     M86  ; ﾊﾟﾚｯﾄ冶具押込LS異常
      ANI     M87  ; ﾅｯﾄﾗﾝﾅｰ部ﾜｰｸ位置決め3LS異常
      ANI     M88  ; ﾅｯﾄﾗﾝﾅｰ部ﾜｰｸ位置決め3ｼﾌﾄLS異常
      ANI     M89  ; ﾅｯﾄﾗﾝﾅｰ部着座確認LS異常
      ANI     M90  ; ﾒｲﾝﾅｯﾄﾗﾝﾅｰLS異常
      ANI     M91  ; ｻﾌﾞﾅｯﾄﾗﾝﾅｰLS異常
      ANI     M92  ; 下流ﾘﾌﾄLS異常
      ANI     M93  ; 引込みﾌﾟｯｼｬｰLS異常
      ANI     M111  ; ﾒｲﾝﾅｯﾄﾗﾝﾅｼｽﾃﾑ異常
      ANI     M112  ; ﾒｲﾝﾅｯﾄﾗﾝﾅ締付異常(ﾄﾙｸ)
      ANI     M113  ; ﾒｲﾝﾅｯﾄﾗﾝﾅ締付異常(角度)
      ANI     M114  ; ｻﾌﾞﾅｯﾄﾗﾝﾅｼｽﾃﾑ異常
      ANI     M115  ; ｻﾌﾞﾅｯﾄﾗﾝﾅ締付異常(ﾄﾙｸ)
      ANI     M116  ; ｻﾌﾞﾅｯﾄﾗﾝﾅ締付異常(角度)
      ANI     M120  ; ID読出し異常
      ANI     M121  ; ID書込み異常
      ANI     T70  ; ﾅｯﾄﾗﾝﾅｰ前ｽﾄｯﾊﾟｰ部ｽﾄｯﾊﾟｰ動作異常
      ANI     T71  ; ﾅｯﾄﾗﾝﾅｰ部ｽﾄｯﾊﾟｰ動作異常
      ANI     T72  ; ﾅｯﾄﾗﾝﾅｰ部位置決め動作異常
      ANI     T73  ; ﾅｯﾄﾗﾝﾅｰ部ｸﾗﾝﾌﾟ1開閉動作異常
      ANI     T74  ; ﾅｯﾄﾗﾝﾅｰ部ｸﾗﾝﾌﾟ1前後動作異常
      ANI     T75  ; ﾅｯﾄﾗﾝﾅｰ部ﾜｰｸ位置決め1動作異常
      ANI     T76  ; ﾊﾟﾚｯﾄ冶具押込動作異常
      ANI     T77  ; ﾅｯﾄﾗﾝﾅｰ部ﾜｰｸ位置決め3動作異常
      ANI     T78  ; ﾅｯﾄﾗﾝﾅｰ部ﾜｰｸ位置決め3ｼﾌﾄ動作異常
      ANI     T79  ; ﾅｯﾄﾗﾝﾅｰ部着座確認動作異常
      ANI     T80  ; ﾒｲﾝﾅｯﾄﾗﾝﾅｰ動作異常
      ANI     T81  ; ｻﾌﾞﾅｯﾄﾗﾝﾅｰ動作異常
      ANI     T82  ; 下流ﾘﾌﾄ動作異常
      ANI     T83  ; 引込みﾌﾟｯｼｬｰ後退動作異常
      ANI     T100  ; ﾒｲﾝﾅｯﾄﾗﾝﾅ ﾀｲﾑｵｰﾊﾞｰ
      ANI     T101  ; ｻﾌﾞﾅｯﾄﾗﾝﾅ ﾀｲﾑｵｰﾊﾞｰ
      ANI     T103  ; 着座詰り異常
      ANI     M117  ; 着座目詰まり異常
      ANI     M118  ; ﾊﾟﾚｯﾄ爪開き異常
      ANI     T104  ; 受渡ｺﾝﾍﾞｱ搬送異常
      ANI     T110  ; ID読出しﾀｲﾑｵｰﾊﾞｰ
      ANI     T111  ; ID書込みﾀｲﾑｵｰﾊﾞｰ
      ANI     C1  ; ﾊﾟﾚｯﾄ着座異常
      ANI     M122  ; IDｺﾝﾄﾛｰﾗｰ異常
      ANI     M195
      ANI     M123
      OUT     M135  ; ﾅｯﾄﾗﾝﾅｰ部異常無
1688  LDI     M100  ; ﾊﾟﾚｯﾄﾌﾟｯｼｬｰ前1ヶ送り部上流LS異常
      ANI     M101  ; ﾊﾟﾚｯﾄﾌﾟｯｼｬｰ前1ヶ送り部下流LS異常
      ANI     M102  ; ﾊﾟﾚｯﾄﾌﾟｯｼｬｰ部ﾌﾟｯｼｬｰLS異常
      ANI     M105  ; 受取ﾘﾌﾄLS異常
      ANI     T90  ; ﾊﾟﾚｯﾄﾌﾟｯｼｬｰ前1ヶ送り上流動作異常
      ANI     T91  ; ﾊﾟﾚｯﾄﾌﾟｯｼｬｰ前1ヶ送り下流動作異常
      ANI     T92  ; ﾊﾟﾚｯﾄﾌﾟｯｼｬｰ部ﾌﾟｯｼｬｰ動作異常
      ANI     T94  ; 上昇ﾘﾌﾀｰ前1ヶ送り下流動作異常
      ANI     T95  ; 受取ﾘﾌﾄ動作異常
      ANI     T106  ; ﾘﾀｰﾝｺﾝﾍﾞｱ1,2,3流れ異常
      OUT     M136  ; ﾘﾀｰﾝｺﾝﾍﾞｱ1,2,3部異常無
1699  LDI     M103  ; 上昇ﾘﾌﾀｰ前1ヶ送り部上流LS異常
      ANI     M104  ; 上昇ﾘﾌﾀｰ前1ヶ送り部下流LS異常
      ANI     M106  ; 受渡ﾘﾌﾄLS異常
      ANI     T93  ; 上昇ﾘﾌﾀｰ前1ヶ送り上流動作異常
      ANI     T96  ; 受渡ﾘﾌﾄ動作異常
      ANI     T107  ; ﾘﾀｰﾝｺﾝﾍﾞｱ4流れ異常
      ANI     M143
      OUT     M137  ; ﾘﾀｰﾝｺﾝﾍﾞｱ4部異常無
1707  LDI     M107  ; 上昇ﾘﾌﾀｰLS異常
      ANI     T97  ; 上昇ﾘﾌﾀｰ動作異常
      ANI     T105  ; 上昇ﾘﾌﾀｰ流れ異常
      OUT     M138  ; 上昇ﾘﾌﾀｰ部異常無
1711  LDI     M23  ; ﾌﾟﾗｸﾞ異常
      ANI     M24  ; ｴｱｰ圧低下
      ANI     M124  ; ｲﾝﾊﾞｰﾀｰ1ｱﾗｰﾑ
      ANI     M125  ; ｲﾝﾊﾞｰﾀｰ2ｱﾗｰﾑ
      ANI     M126  ; ﾘﾀｰﾝｺﾝﾍﾞｱ1ｻｰﾏﾙﾄﾘｯﾌﾟ
      ANI     M127  ; ﾘﾀｰﾝｺﾝﾍﾞｱ2ｻｰﾏﾙﾄﾘｯﾌﾟ
      ANI     M128  ; ﾘﾀｰﾝｺﾝﾍﾞｱ3ｻｰﾏﾙﾄﾘｯﾌﾟ
      ANI     M129  ; ｲﾝﾊﾞｰﾀｰ3ｱﾗｰﾑ
      OUT     M139  ; 非常停止異常無
1720  LDI     M21  ; PC電池異常
      ANI     M22  ; ﾛﾎﾞｯﾄ電池異常
      ANI     T114  ; ｺﾝﾍﾞｱ停止放置異常
      OUT     M140  ; その他異常無
1724  LD      M130  ; ﾛﾎﾞｯﾄ部異常無
      AND     M131  ; M12ﾚｰﾝｽﾄｯｶ部異常無
      AND     M132  ; 中間ﾚｰﾝｽﾄｯｶ部異常無
      AND     M133  ; M10ﾚｰﾝｽﾄｯｶ部異常無
      AND     M134  ; 位置決め部異常無
      AND     M135  ; ﾅｯﾄﾗﾝﾅｰ部異常無
      AND     M136  ; ﾘﾀｰﾝｺﾝﾍﾞｱ1,2,3部異常無
      AND     M138  ; 上昇ﾘﾌﾀｰ部異常無
      AND     M139  ; 非常停止異常無
      OUT     M141  ; 設備停止異常無
1734  LD      M141  ; 設備停止異常無
      AND     M140  ; その他異常無
      ORI     X1  ; ﾋｭｰｽﾞ正常
      OUT     M142  ; 総合異常無
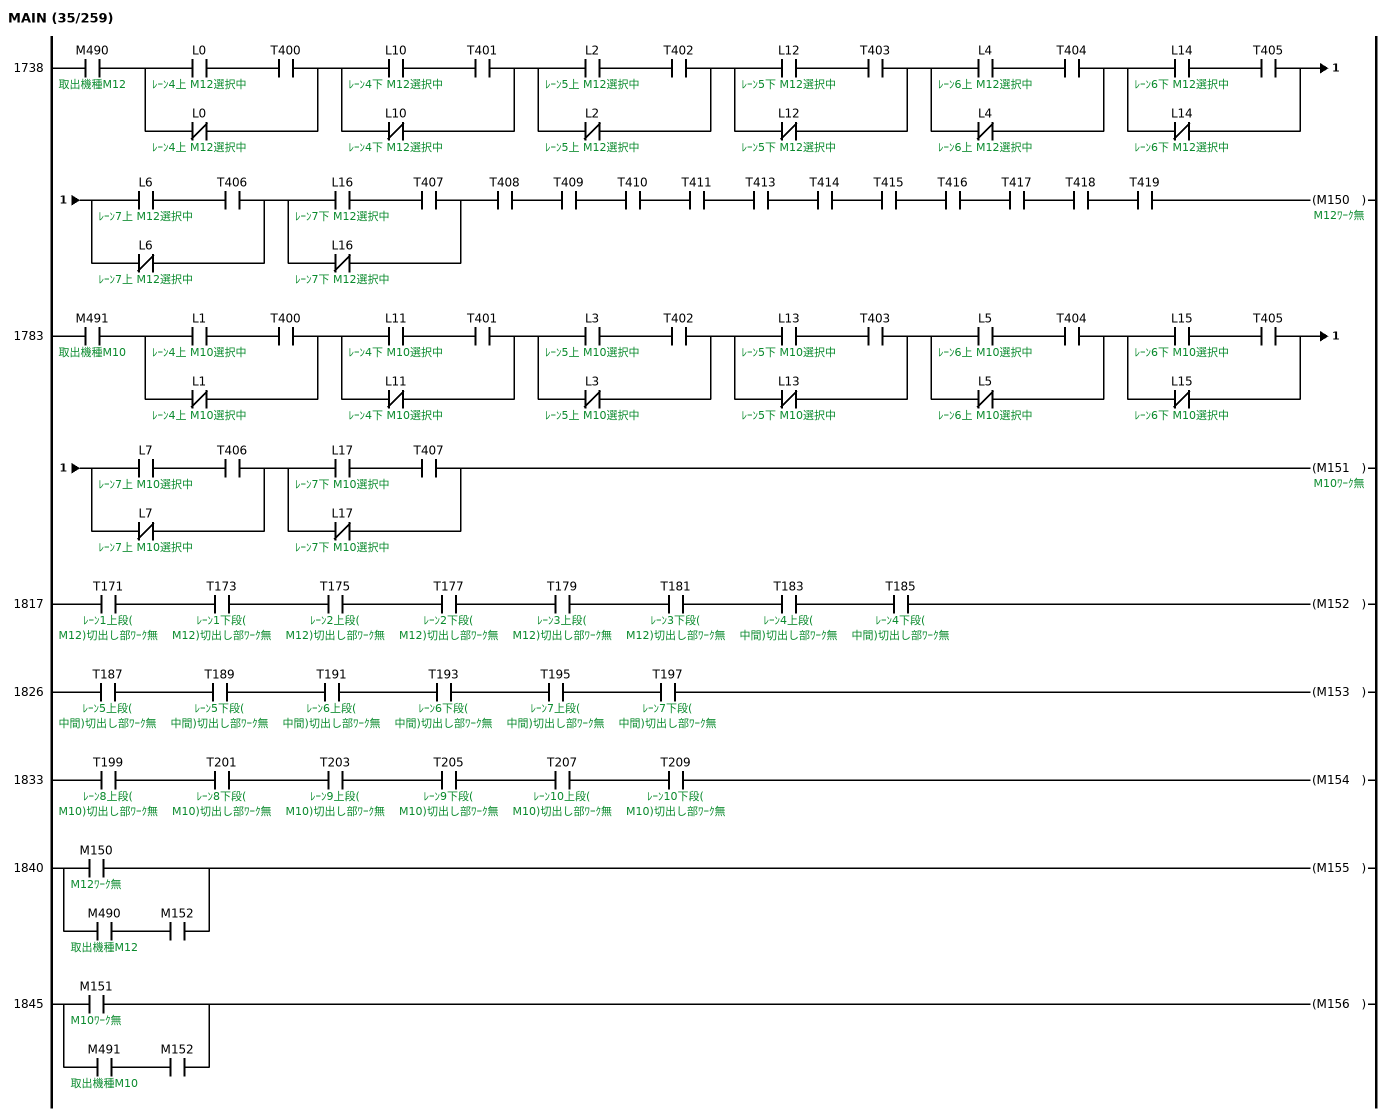
1738  LD      M490  ; 取出機種M12
      LD      L0  ; ﾚｰﾝ4上 M12選択中
      AND     T400
      ORI     L0  ; ﾚｰﾝ4上 M12選択中
      ANB
      LD      L10  ; ﾚｰﾝ4下 M12選択中
      AND     T401
      ORI     L10  ; ﾚｰﾝ4下 M12選択中
      ANB
      LD      L2  ; ﾚｰﾝ5上 M12選択中
      AND     T402
      ORI     L2  ; ﾚｰﾝ5上 M12選択中
      ANB
      LD      L12  ; ﾚｰﾝ5下 M12選択中
      AND     T403
      ORI     L12  ; ﾚｰﾝ5下 M12選択中
      ANB
      LD      L4  ; ﾚｰﾝ6上 M12選択中
      AND     T404
      ORI     L4  ; ﾚｰﾝ6上 M12選択中
      ANB
      LD      L14  ; ﾚｰﾝ6下 M12選択中
      AND     T405
      ORI     L14  ; ﾚｰﾝ6下 M12選択中
      ANB
      LD      L6  ; ﾚｰﾝ7上 M12選択中
      AND     T406
      ORI     L6  ; ﾚｰﾝ7上 M12選択中
      ANB
      LD      L16  ; ﾚｰﾝ7下 M12選択中
      AND     T407
      ORI     L16  ; ﾚｰﾝ7下 M12選択中
      ANB
      AND     T408
      AND     T409
      AND     T410
      AND     T411
      AND     T413
      AND     T414
      AND     T415
      AND     T416
      AND     T417
      AND     T418
      AND     T419
      OUT     M150  ; M12ﾜｰｸ無
1783  LD      M491  ; 取出機種M10
      LD      L1  ; ﾚｰﾝ4上 M10選択中
      AND     T400
      ORI     L1  ; ﾚｰﾝ4上 M10選択中
      ANB
      LD      L11  ; ﾚｰﾝ4下 M10選択中
      AND     T401
      ORI     L11  ; ﾚｰﾝ4下 M10選択中
      ANB
      LD      L3  ; ﾚｰﾝ5上 M10選択中
      AND     T402
      ORI     L3  ; ﾚｰﾝ5上 M10選択中
      ANB
      LD      L13  ; ﾚｰﾝ5下 M10選択中
      AND     T403
      ORI     L13  ; ﾚｰﾝ5下 M10選択中
      ANB
      LD      L5  ; ﾚｰﾝ6上 M10選択中
      AND     T404
      ORI     L5  ; ﾚｰﾝ6上 M10選択中
      ANB
      LD      L15  ; ﾚｰﾝ6下 M10選択中
      AND     T405
      ORI     L15  ; ﾚｰﾝ6下 M10選択中
      ANB
      LD      L7  ; ﾚｰﾝ7上 M10選択中
      AND     T406
      ORI     L7  ; ﾚｰﾝ7上 M10選択中
      ANB
      LD      L17  ; ﾚｰﾝ7下 M10選択中
      AND     T407
      ORI     L17  ; ﾚｰﾝ7下 M10選択中
      ANB
      OUT     M151  ; M10ﾜｰｸ無
1817  LD      T171  ; ﾚｰﾝ1上段(M12)切出し部ﾜｰｸ無
      AND     T173  ; ﾚｰﾝ1下段(M12)切出し部ﾜｰｸ無
      AND     T175  ; ﾚｰﾝ2上段(M12)切出し部ﾜｰｸ無
      AND     T177  ; ﾚｰﾝ2下段(M12)切出し部ﾜｰｸ無
      AND     T179  ; ﾚｰﾝ3上段(M12)切出し部ﾜｰｸ無
      AND     T181  ; ﾚｰﾝ3下段(M12)切出し部ﾜｰｸ無
      AND     T183  ; ﾚｰﾝ4上段(中間)切出し部ﾜｰｸ無
      AND     T185  ; ﾚｰﾝ4下段(中間)切出し部ﾜｰｸ無
      OUT     M152
1826  LD      T187  ; ﾚｰﾝ5上段(中間)切出し部ﾜｰｸ無
      AND     T189  ; ﾚｰﾝ5下段(中間)切出し部ﾜｰｸ無
      AND     T191  ; ﾚｰﾝ6上段(中間)切出し部ﾜｰｸ無
      AND     T193  ; ﾚｰﾝ6下段(中間)切出し部ﾜｰｸ無
      AND     T195  ; ﾚｰﾝ7上段(中間)切出し部ﾜｰｸ無
      AND     T197  ; ﾚｰﾝ7下段(中間)切出し部ﾜｰｸ無
      OUT     M153
1833  LD      T199  ; ﾚｰﾝ8上段(M10)切出し部ﾜｰｸ無
      AND     T201  ; ﾚｰﾝ8下段(M10)切出し部ﾜｰｸ無
      AND     T203  ; ﾚｰﾝ9上段(M10)切出し部ﾜｰｸ無
      AND     T205  ; ﾚｰﾝ9下段(M10)切出し部ﾜｰｸ無
      AND     T207  ; ﾚｰﾝ10上段(M10)切出し部ﾜｰｸ無
      AND     T209  ; ﾚｰﾝ10下段(M10)切出し部ﾜｰｸ無
      OUT     M154
1840  LD      M150  ; M12ﾜｰｸ無
      LD      M490  ; 取出機種M12
      AND     M152
      ORB
      OUT     M155
1845  LD      M151  ; M10ﾜｰｸ無
      LD      M491  ; 取出機種M10
      AND     M152
      ORB
      OUT     M156
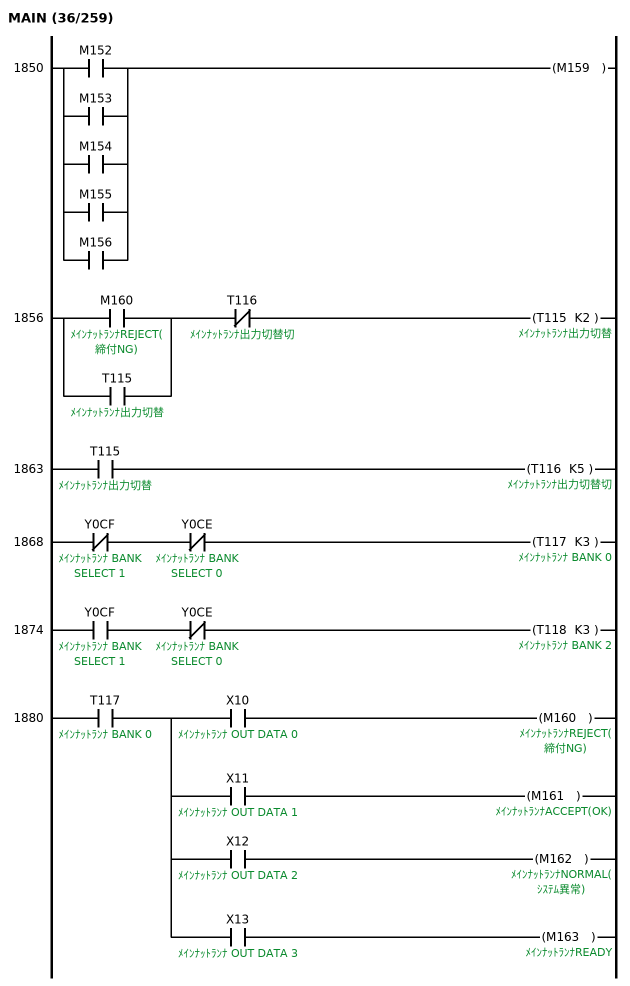
1850  LD      M152
      OR      M153
      OR      M154
      OR      M155
      OR      M156
      OUT     M159
1856  LD      M160  ; ﾒｲﾝﾅｯﾄﾗﾝﾅREJECT(締付NG)
      OR      T115  ; ﾒｲﾝﾅｯﾄﾗﾝﾅ出力切替
      ANI     T116  ; ﾒｲﾝﾅｯﾄﾗﾝﾅ出力切替切
      OUT     T115 K2  ; ﾒｲﾝﾅｯﾄﾗﾝﾅ出力切替
1863  LD      T115  ; ﾒｲﾝﾅｯﾄﾗﾝﾅ出力切替
      OUT     T116 K5  ; ﾒｲﾝﾅｯﾄﾗﾝﾅ出力切替切
1868  LDI     Y0CF  ; ﾒｲﾝﾅｯﾄﾗﾝﾅ BANK SELECT 1
      ANI     Y0CE  ; ﾒｲﾝﾅｯﾄﾗﾝﾅ BANK SELECT 0
      OUT     T117 K3  ; ﾒｲﾝﾅｯﾄﾗﾝﾅ BANK 0
1874  LD      Y0CF  ; ﾒｲﾝﾅｯﾄﾗﾝﾅ BANK SELECT 1
      ANI     Y0CE  ; ﾒｲﾝﾅｯﾄﾗﾝﾅ BANK SELECT 0
      OUT     T118 K3  ; ﾒｲﾝﾅｯﾄﾗﾝﾅ BANK 2
1880  LD      T117  ; ﾒｲﾝﾅｯﾄﾗﾝﾅ BANK 0
      MPS
      AND     X10  ; ﾒｲﾝﾅｯﾄﾗﾝﾅ OUT DATA 0
      OUT     M160  ; ﾒｲﾝﾅｯﾄﾗﾝﾅREJECT(締付NG)
      MRD
      AND     X11  ; ﾒｲﾝﾅｯﾄﾗﾝﾅ OUT DATA 1
      OUT     M161  ; ﾒｲﾝﾅｯﾄﾗﾝﾅACCEPT(OK)
      MRD
      AND     X12  ; ﾒｲﾝﾅｯﾄﾗﾝﾅ OUT DATA 2
      OUT     M162  ; ﾒｲﾝﾅｯﾄﾗﾝﾅNORMAL(ｼｽﾃﾑ異常)
      MPP
      AND     X13  ; ﾒｲﾝﾅｯﾄﾗﾝﾅ OUT DATA 3
      OUT     M163  ; ﾒｲﾝﾅｯﾄﾗﾝﾅREADY
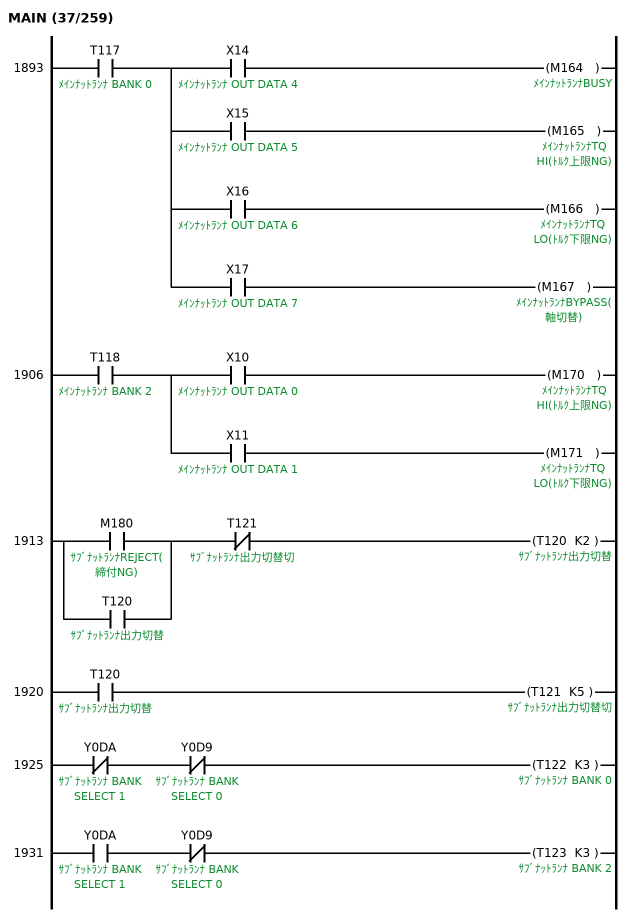
1893  LD      T117  ; ﾒｲﾝﾅｯﾄﾗﾝﾅ BANK 0
      MPS
      AND     X14  ; ﾒｲﾝﾅｯﾄﾗﾝﾅ OUT DATA 4
      OUT     M164  ; ﾒｲﾝﾅｯﾄﾗﾝﾅBUSY
      MRD
      AND     X15  ; ﾒｲﾝﾅｯﾄﾗﾝﾅ OUT DATA 5
      OUT     M165  ; ﾒｲﾝﾅｯﾄﾗﾝﾅTQ HI(ﾄﾙｸ上限NG)
      MRD
      AND     X16  ; ﾒｲﾝﾅｯﾄﾗﾝﾅ OUT DATA 6
      OUT     M166  ; ﾒｲﾝﾅｯﾄﾗﾝﾅTQ LO(ﾄﾙｸ下限NG)
      MPP
      AND     X17  ; ﾒｲﾝﾅｯﾄﾗﾝﾅ OUT DATA 7
      OUT     M167  ; ﾒｲﾝﾅｯﾄﾗﾝﾅBYPASS(軸切替)
1906  LD      T118  ; ﾒｲﾝﾅｯﾄﾗﾝﾅ BANK 2
      MPS
      AND     X10  ; ﾒｲﾝﾅｯﾄﾗﾝﾅ OUT DATA 0
      OUT     M170  ; ﾒｲﾝﾅｯﾄﾗﾝﾅTQ HI(ﾄﾙｸ上限NG)
      MPP
      AND     X11  ; ﾒｲﾝﾅｯﾄﾗﾝﾅ OUT DATA 1
      OUT     M171  ; ﾒｲﾝﾅｯﾄﾗﾝﾅTQ LO(ﾄﾙｸ下限NG)
1913  LD      M180  ; ｻﾌﾞﾅｯﾄﾗﾝﾅREJECT(締付NG)
      OR      T120  ; ｻﾌﾞﾅｯﾄﾗﾝﾅ出力切替
      ANI     T121  ; ｻﾌﾞﾅｯﾄﾗﾝﾅ出力切替切
      OUT     T120 K2  ; ｻﾌﾞﾅｯﾄﾗﾝﾅ出力切替
1920  LD      T120  ; ｻﾌﾞﾅｯﾄﾗﾝﾅ出力切替
      OUT     T121 K5  ; ｻﾌﾞﾅｯﾄﾗﾝﾅ出力切替切
1925  LDI     Y0DA  ; ｻﾌﾞﾅｯﾄﾗﾝﾅ BANK SELECT 1
      ANI     Y0D9  ; ｻﾌﾞﾅｯﾄﾗﾝﾅ BANK SELECT 0
      OUT     T122 K3  ; ｻﾌﾞﾅｯﾄﾗﾝﾅ BANK 0
1931  LD      Y0DA  ; ｻﾌﾞﾅｯﾄﾗﾝﾅ BANK SELECT 1
      ANI     Y0D9  ; ｻﾌﾞﾅｯﾄﾗﾝﾅ BANK SELECT 0
      OUT     T123 K3  ; ｻﾌﾞﾅｯﾄﾗﾝﾅ BANK 2
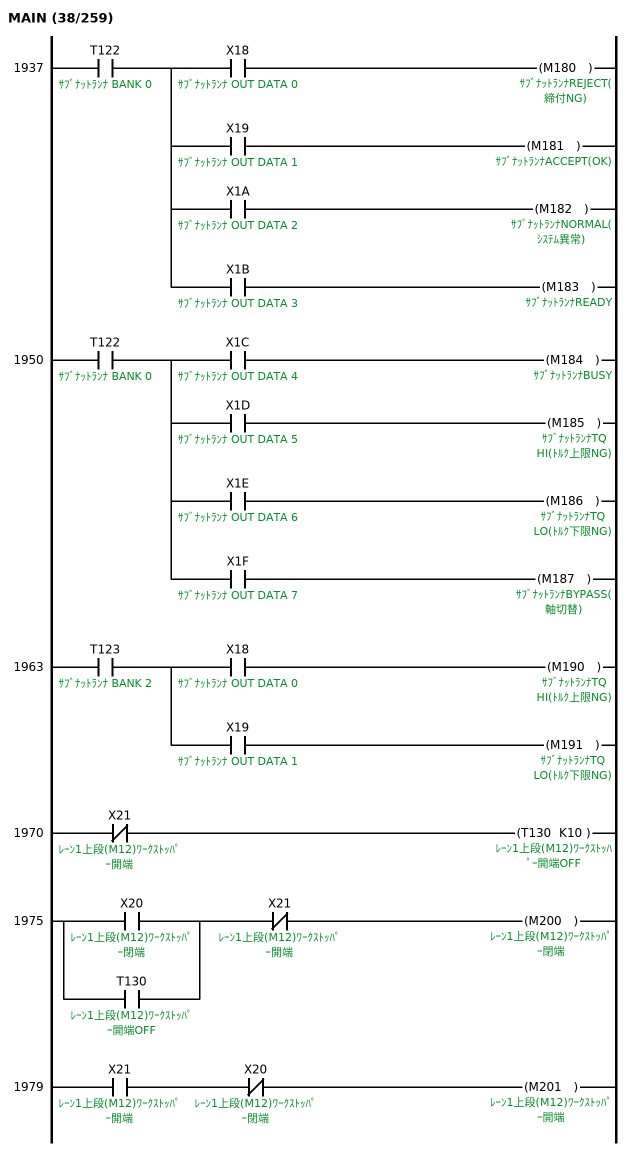
1937  LD      T122  ; ｻﾌﾞﾅｯﾄﾗﾝﾅ BANK 0
      MPS
      AND     X18  ; ｻﾌﾞﾅｯﾄﾗﾝﾅ OUT DATA 0
      OUT     M180  ; ｻﾌﾞﾅｯﾄﾗﾝﾅREJECT(締付NG)
      MRD
      AND     X19  ; ｻﾌﾞﾅｯﾄﾗﾝﾅ OUT DATA 1
      OUT     M181  ; ｻﾌﾞﾅｯﾄﾗﾝﾅACCEPT(OK)
      MRD
      AND     X1A  ; ｻﾌﾞﾅｯﾄﾗﾝﾅ OUT DATA 2
      OUT     M182  ; ｻﾌﾞﾅｯﾄﾗﾝﾅNORMAL(ｼｽﾃﾑ異常)
      MPP
      AND     X1B  ; ｻﾌﾞﾅｯﾄﾗﾝﾅ OUT DATA 3
      OUT     M183  ; ｻﾌﾞﾅｯﾄﾗﾝﾅREADY
1950  LD      T122  ; ｻﾌﾞﾅｯﾄﾗﾝﾅ BANK 0
      MPS
      AND     X1C  ; ｻﾌﾞﾅｯﾄﾗﾝﾅ OUT DATA 4
      OUT     M184  ; ｻﾌﾞﾅｯﾄﾗﾝﾅBUSY
      MRD
      AND     X1D  ; ｻﾌﾞﾅｯﾄﾗﾝﾅ OUT DATA 5
      OUT     M185  ; ｻﾌﾞﾅｯﾄﾗﾝﾅTQ HI(ﾄﾙｸ上限NG)
      MRD
      AND     X1E  ; ｻﾌﾞﾅｯﾄﾗﾝﾅ OUT DATA 6
      OUT     M186  ; ｻﾌﾞﾅｯﾄﾗﾝﾅTQ LO(ﾄﾙｸ下限NG)
      MPP
      AND     X1F  ; ｻﾌﾞﾅｯﾄﾗﾝﾅ OUT DATA 7
      OUT     M187  ; ｻﾌﾞﾅｯﾄﾗﾝﾅBYPASS(軸切替)
1963  LD      T123  ; ｻﾌﾞﾅｯﾄﾗﾝﾅ BANK 2
      MPS
      AND     X18  ; ｻﾌﾞﾅｯﾄﾗﾝﾅ OUT DATA 0
      OUT     M190  ; ｻﾌﾞﾅｯﾄﾗﾝﾅTQ HI(ﾄﾙｸ上限NG)
      MPP
      AND     X19  ; ｻﾌﾞﾅｯﾄﾗﾝﾅ OUT DATA 1
      OUT     M191  ; ｻﾌﾞﾅｯﾄﾗﾝﾅTQ LO(ﾄﾙｸ下限NG)
1970  LDI     X21  ; ﾚｰﾝ1上段(M12)ﾜｰｸｽﾄｯﾊﾟｰ開端
      OUT     T130 K10  ; ﾚｰﾝ1上段(M12)ﾜｰｸｽﾄｯﾊﾟｰ開端OFF
1975  LD      X20  ; ﾚｰﾝ1上段(M12)ﾜｰｸｽﾄｯﾊﾟｰ閉端
      OR      T130  ; ﾚｰﾝ1上段(M12)ﾜｰｸｽﾄｯﾊﾟｰ開端OFF
      ANI     X21  ; ﾚｰﾝ1上段(M12)ﾜｰｸｽﾄｯﾊﾟｰ開端
      OUT     M200  ; ﾚｰﾝ1上段(M12)ﾜｰｸｽﾄｯﾊﾟｰ閉端
1979  LD      X21  ; ﾚｰﾝ1上段(M12)ﾜｰｸｽﾄｯﾊﾟｰ開端
      ANI     X20  ; ﾚｰﾝ1上段(M12)ﾜｰｸｽﾄｯﾊﾟｰ閉端
      OUT     M201  ; ﾚｰﾝ1上段(M12)ﾜｰｸｽﾄｯﾊﾟｰ開端
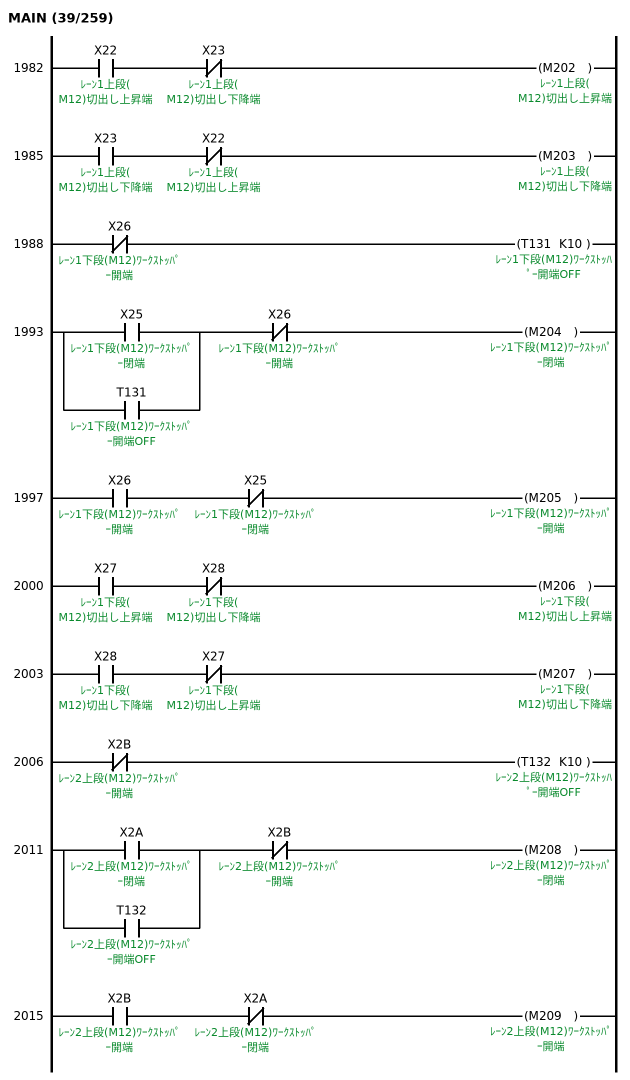
1982  LD      X22  ; ﾚｰﾝ1上段(M12)切出し上昇端
      ANI     X23  ; ﾚｰﾝ1上段(M12)切出し下降端
      OUT     M202  ; ﾚｰﾝ1上段(M12)切出し上昇端
1985  LD      X23  ; ﾚｰﾝ1上段(M12)切出し下降端
      ANI     X22  ; ﾚｰﾝ1上段(M12)切出し上昇端
      OUT     M203  ; ﾚｰﾝ1上段(M12)切出し下降端
1988  LDI     X26  ; ﾚｰﾝ1下段(M12)ﾜｰｸｽﾄｯﾊﾟｰ開端
      OUT     T131 K10  ; ﾚｰﾝ1下段(M12)ﾜｰｸｽﾄｯﾊﾟｰ開端OFF
1993  LD      X25  ; ﾚｰﾝ1下段(M12)ﾜｰｸｽﾄｯﾊﾟｰ閉端
      OR      T131  ; ﾚｰﾝ1下段(M12)ﾜｰｸｽﾄｯﾊﾟｰ開端OFF
      ANI     X26  ; ﾚｰﾝ1下段(M12)ﾜｰｸｽﾄｯﾊﾟｰ開端
      OUT     M204  ; ﾚｰﾝ1下段(M12)ﾜｰｸｽﾄｯﾊﾟｰ閉端
1997  LD      X26  ; ﾚｰﾝ1下段(M12)ﾜｰｸｽﾄｯﾊﾟｰ開端
      ANI     X25  ; ﾚｰﾝ1下段(M12)ﾜｰｸｽﾄｯﾊﾟｰ閉端
      OUT     M205  ; ﾚｰﾝ1下段(M12)ﾜｰｸｽﾄｯﾊﾟｰ開端
2000  LD      X27  ; ﾚｰﾝ1下段(M12)切出し上昇端
      ANI     X28  ; ﾚｰﾝ1下段(M12)切出し下降端
      OUT     M206  ; ﾚｰﾝ1下段(M12)切出し上昇端
2003  LD      X28  ; ﾚｰﾝ1下段(M12)切出し下降端
      ANI     X27  ; ﾚｰﾝ1下段(M12)切出し上昇端
      OUT     M207  ; ﾚｰﾝ1下段(M12)切出し下降端
2006  LDI     X2B  ; ﾚｰﾝ2上段(M12)ﾜｰｸｽﾄｯﾊﾟｰ開端
      OUT     T132 K10  ; ﾚｰﾝ2上段(M12)ﾜｰｸｽﾄｯﾊﾟｰ開端OFF
2011  LD      X2A  ; ﾚｰﾝ2上段(M12)ﾜｰｸｽﾄｯﾊﾟｰ閉端
      OR      T132  ; ﾚｰﾝ2上段(M12)ﾜｰｸｽﾄｯﾊﾟｰ開端OFF
      ANI     X2B  ; ﾚｰﾝ2上段(M12)ﾜｰｸｽﾄｯﾊﾟｰ開端
      OUT     M208  ; ﾚｰﾝ2上段(M12)ﾜｰｸｽﾄｯﾊﾟｰ閉端
2015  LD      X2B  ; ﾚｰﾝ2上段(M12)ﾜｰｸｽﾄｯﾊﾟｰ開端
      ANI     X2A  ; ﾚｰﾝ2上段(M12)ﾜｰｸｽﾄｯﾊﾟｰ閉端
      OUT     M209  ; ﾚｰﾝ2上段(M12)ﾜｰｸｽﾄｯﾊﾟｰ開端
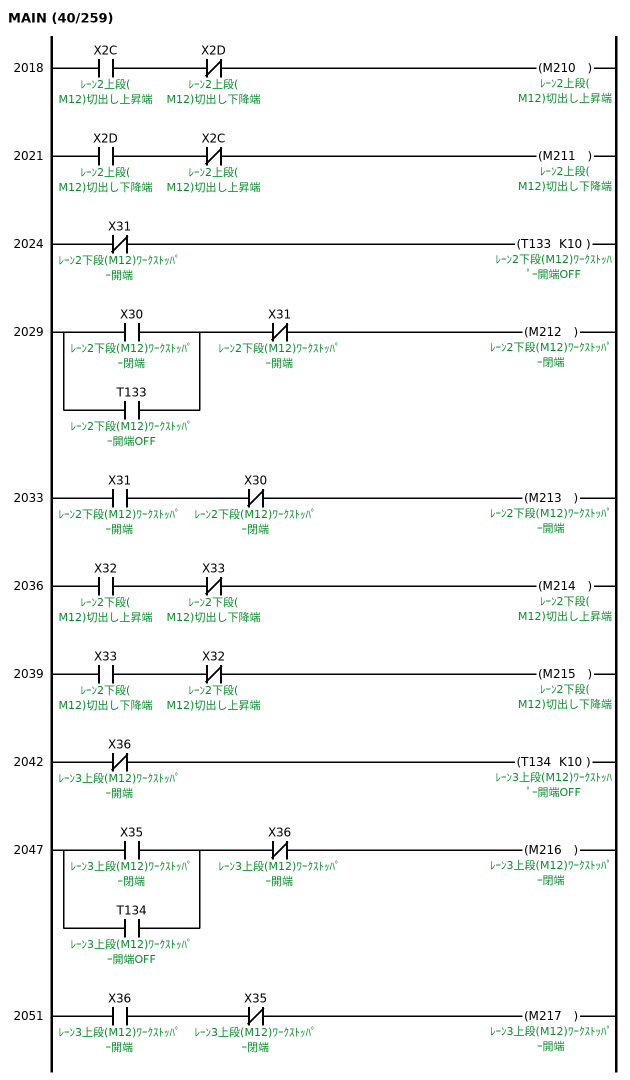
2018  LD      X2C  ; ﾚｰﾝ2上段(M12)切出し上昇端
      ANI     X2D  ; ﾚｰﾝ2上段(M12)切出し下降端
      OUT     M210  ; ﾚｰﾝ2上段(M12)切出し上昇端
2021  LD      X2D  ; ﾚｰﾝ2上段(M12)切出し下降端
      ANI     X2C  ; ﾚｰﾝ2上段(M12)切出し上昇端
      OUT     M211  ; ﾚｰﾝ2上段(M12)切出し下降端
2024  LDI     X31  ; ﾚｰﾝ2下段(M12)ﾜｰｸｽﾄｯﾊﾟｰ開端
      OUT     T133 K10  ; ﾚｰﾝ2下段(M12)ﾜｰｸｽﾄｯﾊﾟｰ開端OFF
2029  LD      X30  ; ﾚｰﾝ2下段(M12)ﾜｰｸｽﾄｯﾊﾟｰ閉端
      OR      T133  ; ﾚｰﾝ2下段(M12)ﾜｰｸｽﾄｯﾊﾟｰ開端OFF
      ANI     X31  ; ﾚｰﾝ2下段(M12)ﾜｰｸｽﾄｯﾊﾟｰ開端
      OUT     M212  ; ﾚｰﾝ2下段(M12)ﾜｰｸｽﾄｯﾊﾟｰ閉端
2033  LD      X31  ; ﾚｰﾝ2下段(M12)ﾜｰｸｽﾄｯﾊﾟｰ開端
      ANI     X30  ; ﾚｰﾝ2下段(M12)ﾜｰｸｽﾄｯﾊﾟｰ閉端
      OUT     M213  ; ﾚｰﾝ2下段(M12)ﾜｰｸｽﾄｯﾊﾟｰ開端
2036  LD      X32  ; ﾚｰﾝ2下段(M12)切出し上昇端
      ANI     X33  ; ﾚｰﾝ2下段(M12)切出し下降端
      OUT     M214  ; ﾚｰﾝ2下段(M12)切出し上昇端
2039  LD      X33  ; ﾚｰﾝ2下段(M12)切出し下降端
      ANI     X32  ; ﾚｰﾝ2下段(M12)切出し上昇端
      OUT     M215  ; ﾚｰﾝ2下段(M12)切出し下降端
2042  LDI     X36  ; ﾚｰﾝ3上段(M12)ﾜｰｸｽﾄｯﾊﾟｰ開端
      OUT     T134 K10  ; ﾚｰﾝ3上段(M12)ﾜｰｸｽﾄｯﾊﾟｰ開端OFF
2047  LD      X35  ; ﾚｰﾝ3上段(M12)ﾜｰｸｽﾄｯﾊﾟｰ閉端
      OR      T134  ; ﾚｰﾝ3上段(M12)ﾜｰｸｽﾄｯﾊﾟｰ開端OFF
      ANI     X36  ; ﾚｰﾝ3上段(M12)ﾜｰｸｽﾄｯﾊﾟｰ開端
      OUT     M216  ; ﾚｰﾝ3上段(M12)ﾜｰｸｽﾄｯﾊﾟｰ閉端
2051  LD      X36  ; ﾚｰﾝ3上段(M12)ﾜｰｸｽﾄｯﾊﾟｰ開端
      ANI     X35  ; ﾚｰﾝ3上段(M12)ﾜｰｸｽﾄｯﾊﾟｰ閉端
      OUT     M217  ; ﾚｰﾝ3上段(M12)ﾜｰｸｽﾄｯﾊﾟｰ開端
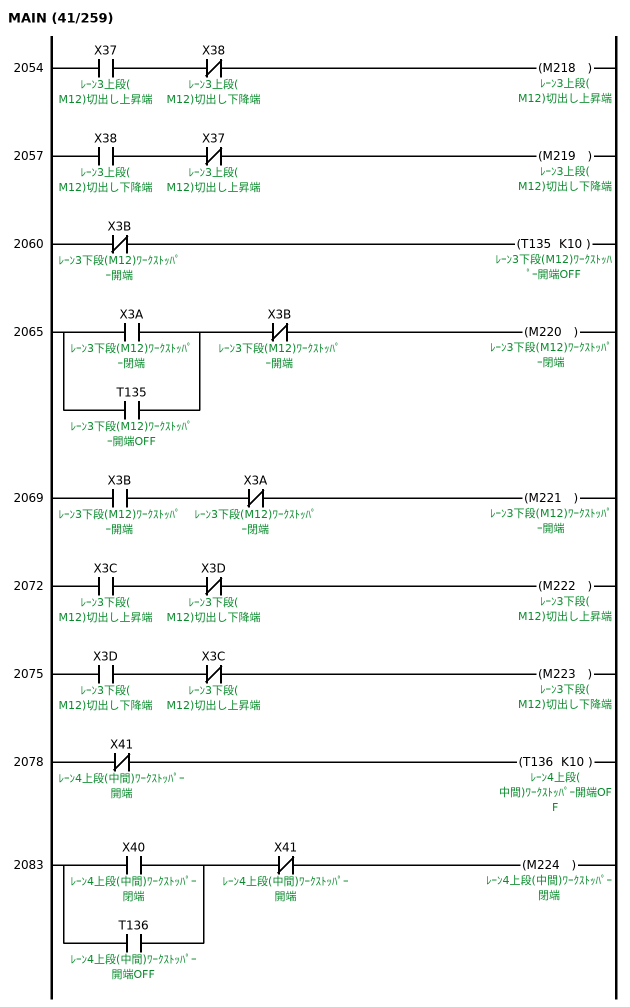
2054  LD      X37  ; ﾚｰﾝ3上段(M12)切出し上昇端
      ANI     X38  ; ﾚｰﾝ3上段(M12)切出し下降端
      OUT     M218  ; ﾚｰﾝ3上段(M12)切出し上昇端
2057  LD      X38  ; ﾚｰﾝ3上段(M12)切出し下降端
      ANI     X37  ; ﾚｰﾝ3上段(M12)切出し上昇端
      OUT     M219  ; ﾚｰﾝ3上段(M12)切出し下降端
2060  LDI     X3B  ; ﾚｰﾝ3下段(M12)ﾜｰｸｽﾄｯﾊﾟｰ開端
      OUT     T135 K10  ; ﾚｰﾝ3下段(M12)ﾜｰｸｽﾄｯﾊﾟｰ開端OFF
2065  LD      X3A  ; ﾚｰﾝ3下段(M12)ﾜｰｸｽﾄｯﾊﾟｰ閉端
      OR      T135  ; ﾚｰﾝ3下段(M12)ﾜｰｸｽﾄｯﾊﾟｰ開端OFF
      ANI     X3B  ; ﾚｰﾝ3下段(M12)ﾜｰｸｽﾄｯﾊﾟｰ開端
      OUT     M220  ; ﾚｰﾝ3下段(M12)ﾜｰｸｽﾄｯﾊﾟｰ閉端
2069  LD      X3B  ; ﾚｰﾝ3下段(M12)ﾜｰｸｽﾄｯﾊﾟｰ開端
      ANI     X3A  ; ﾚｰﾝ3下段(M12)ﾜｰｸｽﾄｯﾊﾟｰ閉端
      OUT     M221  ; ﾚｰﾝ3下段(M12)ﾜｰｸｽﾄｯﾊﾟｰ開端
2072  LD      X3C  ; ﾚｰﾝ3下段(M12)切出し上昇端
      ANI     X3D  ; ﾚｰﾝ3下段(M12)切出し下降端
      OUT     M222  ; ﾚｰﾝ3下段(M12)切出し上昇端
2075  LD      X3D  ; ﾚｰﾝ3下段(M12)切出し下降端
      ANI     X3C  ; ﾚｰﾝ3下段(M12)切出し上昇端
      OUT     M223  ; ﾚｰﾝ3下段(M12)切出し下降端
2078  LDI     X41  ; ﾚｰﾝ4上段(中間)ﾜｰｸｽﾄｯﾊﾟｰ開端
      OUT     T136 K10  ; ﾚｰﾝ4上段(中間)ﾜｰｸｽﾄｯﾊﾟｰ開端OFF
2083  LD      X40  ; ﾚｰﾝ4上段(中間)ﾜｰｸｽﾄｯﾊﾟｰ閉端
      OR      T136  ; ﾚｰﾝ4上段(中間)ﾜｰｸｽﾄｯﾊﾟｰ開端OFF
      ANI     X41  ; ﾚｰﾝ4上段(中間)ﾜｰｸｽﾄｯﾊﾟｰ開端
      OUT     M224  ; ﾚｰﾝ4上段(中間)ﾜｰｸｽﾄｯﾊﾟｰ閉端
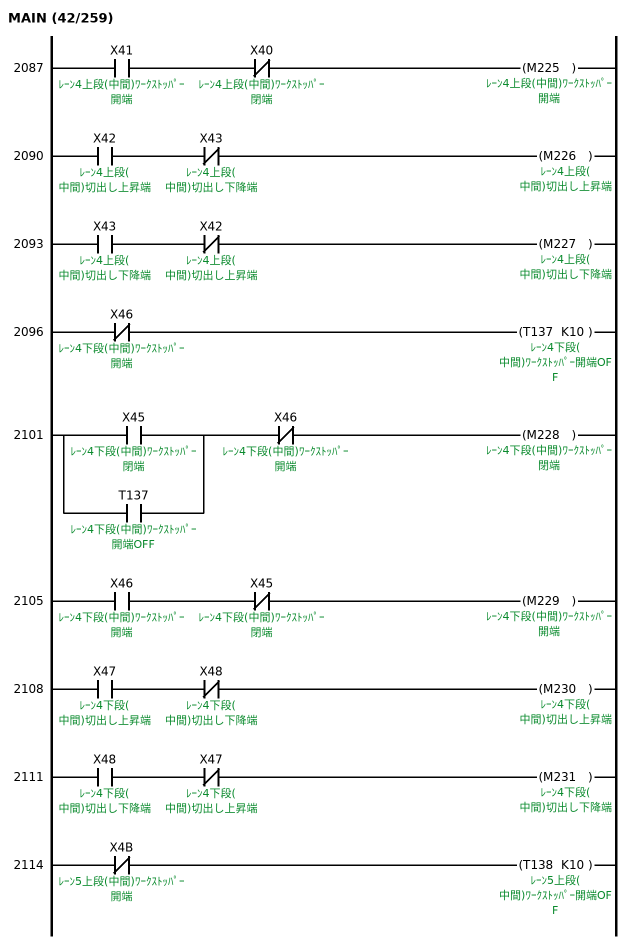
2087  LD      X41  ; ﾚｰﾝ4上段(中間)ﾜｰｸｽﾄｯﾊﾟｰ開端
      ANI     X40  ; ﾚｰﾝ4上段(中間)ﾜｰｸｽﾄｯﾊﾟｰ閉端
      OUT     M225  ; ﾚｰﾝ4上段(中間)ﾜｰｸｽﾄｯﾊﾟｰ開端
2090  LD      X42  ; ﾚｰﾝ4上段(中間)切出し上昇端
      ANI     X43  ; ﾚｰﾝ4上段(中間)切出し下降端
      OUT     M226  ; ﾚｰﾝ4上段(中間)切出し上昇端
2093  LD      X43  ; ﾚｰﾝ4上段(中間)切出し下降端
      ANI     X42  ; ﾚｰﾝ4上段(中間)切出し上昇端
      OUT     M227  ; ﾚｰﾝ4上段(中間)切出し下降端
2096  LDI     X46  ; ﾚｰﾝ4下段(中間)ﾜｰｸｽﾄｯﾊﾟｰ開端
      OUT     T137 K10  ; ﾚｰﾝ4下段(中間)ﾜｰｸｽﾄｯﾊﾟｰ開端OFF
2101  LD      X45  ; ﾚｰﾝ4下段(中間)ﾜｰｸｽﾄｯﾊﾟｰ閉端
      OR      T137  ; ﾚｰﾝ4下段(中間)ﾜｰｸｽﾄｯﾊﾟｰ開端OFF
      ANI     X46  ; ﾚｰﾝ4下段(中間)ﾜｰｸｽﾄｯﾊﾟｰ開端
      OUT     M228  ; ﾚｰﾝ4下段(中間)ﾜｰｸｽﾄｯﾊﾟｰ閉端
2105  LD      X46  ; ﾚｰﾝ4下段(中間)ﾜｰｸｽﾄｯﾊﾟｰ開端
      ANI     X45  ; ﾚｰﾝ4下段(中間)ﾜｰｸｽﾄｯﾊﾟｰ閉端
      OUT     M229  ; ﾚｰﾝ4下段(中間)ﾜｰｸｽﾄｯﾊﾟｰ開端
2108  LD      X47  ; ﾚｰﾝ4下段(中間)切出し上昇端
      ANI     X48  ; ﾚｰﾝ4下段(中間)切出し下降端
      OUT     M230  ; ﾚｰﾝ4下段(中間)切出し上昇端
2111  LD      X48  ; ﾚｰﾝ4下段(中間)切出し下降端
      ANI     X47  ; ﾚｰﾝ4下段(中間)切出し上昇端
      OUT     M231  ; ﾚｰﾝ4下段(中間)切出し下降端
2114  LDI     X4B  ; ﾚｰﾝ5上段(中間)ﾜｰｸｽﾄｯﾊﾟｰ開端
      OUT     T138 K10  ; ﾚｰﾝ5上段(中間)ﾜｰｸｽﾄｯﾊﾟｰ開端OFF
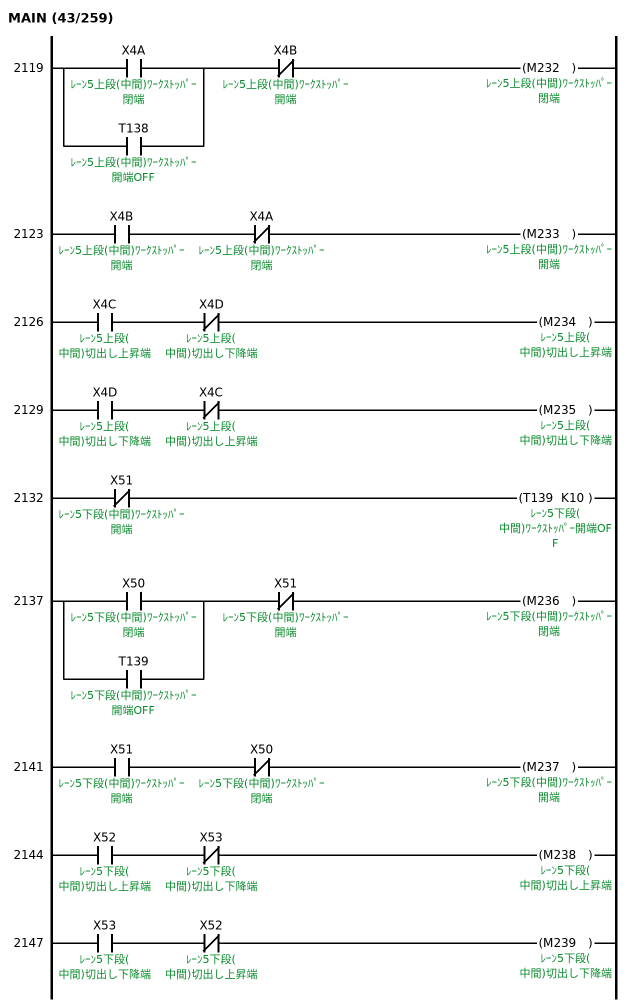
2119  LD      X4A  ; ﾚｰﾝ5上段(中間)ﾜｰｸｽﾄｯﾊﾟｰ閉端
      OR      T138  ; ﾚｰﾝ5上段(中間)ﾜｰｸｽﾄｯﾊﾟｰ開端OFF
      ANI     X4B  ; ﾚｰﾝ5上段(中間)ﾜｰｸｽﾄｯﾊﾟｰ開端
      OUT     M232  ; ﾚｰﾝ5上段(中間)ﾜｰｸｽﾄｯﾊﾟｰ閉端
2123  LD      X4B  ; ﾚｰﾝ5上段(中間)ﾜｰｸｽﾄｯﾊﾟｰ開端
      ANI     X4A  ; ﾚｰﾝ5上段(中間)ﾜｰｸｽﾄｯﾊﾟｰ閉端
      OUT     M233  ; ﾚｰﾝ5上段(中間)ﾜｰｸｽﾄｯﾊﾟｰ開端
2126  LD      X4C  ; ﾚｰﾝ5上段(中間)切出し上昇端
      ANI     X4D  ; ﾚｰﾝ5上段(中間)切出し下降端
      OUT     M234  ; ﾚｰﾝ5上段(中間)切出し上昇端
2129  LD      X4D  ; ﾚｰﾝ5上段(中間)切出し下降端
      ANI     X4C  ; ﾚｰﾝ5上段(中間)切出し上昇端
      OUT     M235  ; ﾚｰﾝ5上段(中間)切出し下降端
2132  LDI     X51  ; ﾚｰﾝ5下段(中間)ﾜｰｸｽﾄｯﾊﾟｰ開端
      OUT     T139 K10  ; ﾚｰﾝ5下段(中間)ﾜｰｸｽﾄｯﾊﾟｰ開端OFF
2137  LD      X50  ; ﾚｰﾝ5下段(中間)ﾜｰｸｽﾄｯﾊﾟｰ閉端
      OR      T139  ; ﾚｰﾝ5下段(中間)ﾜｰｸｽﾄｯﾊﾟｰ開端OFF
      ANI     X51  ; ﾚｰﾝ5下段(中間)ﾜｰｸｽﾄｯﾊﾟｰ開端
      OUT     M236  ; ﾚｰﾝ5下段(中間)ﾜｰｸｽﾄｯﾊﾟｰ閉端
2141  LD      X51  ; ﾚｰﾝ5下段(中間)ﾜｰｸｽﾄｯﾊﾟｰ開端
      ANI     X50  ; ﾚｰﾝ5下段(中間)ﾜｰｸｽﾄｯﾊﾟｰ閉端
      OUT     M237  ; ﾚｰﾝ5下段(中間)ﾜｰｸｽﾄｯﾊﾟｰ開端
2144  LD      X52  ; ﾚｰﾝ5下段(中間)切出し上昇端
      ANI     X53  ; ﾚｰﾝ5下段(中間)切出し下降端
      OUT     M238  ; ﾚｰﾝ5下段(中間)切出し上昇端
2147  LD      X53  ; ﾚｰﾝ5下段(中間)切出し下降端
      ANI     X52  ; ﾚｰﾝ5下段(中間)切出し上昇端
      OUT     M239  ; ﾚｰﾝ5下段(中間)切出し下降端
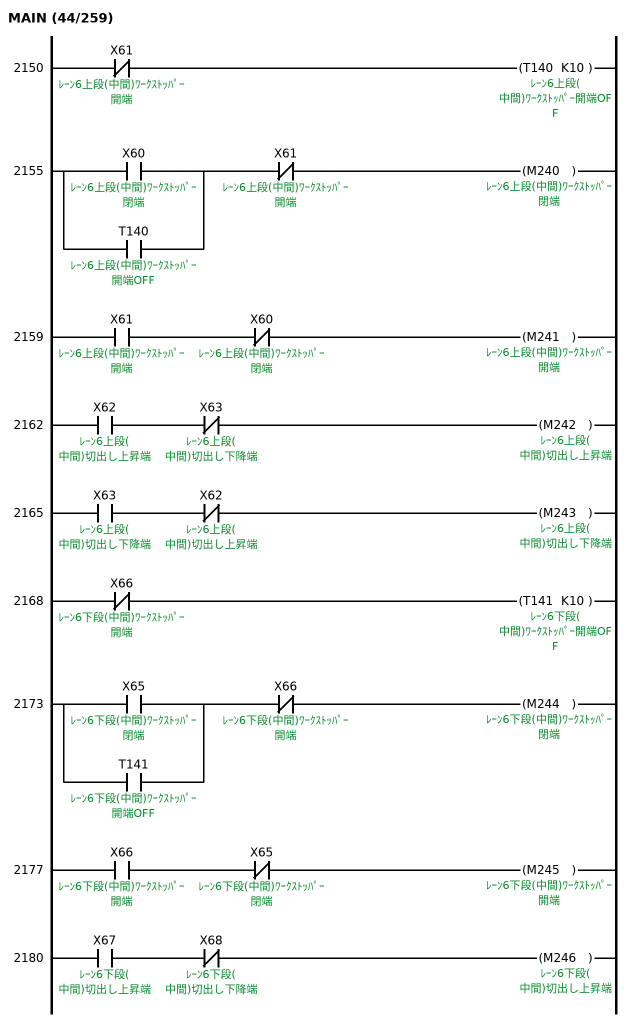
2150  LDI     X61  ; ﾚｰﾝ6上段(中間)ﾜｰｸｽﾄｯﾊﾟｰ開端
      OUT     T140 K10  ; ﾚｰﾝ6上段(中間)ﾜｰｸｽﾄｯﾊﾟｰ開端OFF
2155  LD      X60  ; ﾚｰﾝ6上段(中間)ﾜｰｸｽﾄｯﾊﾟｰ閉端
      OR      T140  ; ﾚｰﾝ6上段(中間)ﾜｰｸｽﾄｯﾊﾟｰ開端OFF
      ANI     X61  ; ﾚｰﾝ6上段(中間)ﾜｰｸｽﾄｯﾊﾟｰ開端
      OUT     M240  ; ﾚｰﾝ6上段(中間)ﾜｰｸｽﾄｯﾊﾟｰ閉端
2159  LD      X61  ; ﾚｰﾝ6上段(中間)ﾜｰｸｽﾄｯﾊﾟｰ開端
      ANI     X60  ; ﾚｰﾝ6上段(中間)ﾜｰｸｽﾄｯﾊﾟｰ閉端
      OUT     M241  ; ﾚｰﾝ6上段(中間)ﾜｰｸｽﾄｯﾊﾟｰ開端
2162  LD      X62  ; ﾚｰﾝ6上段(中間)切出し上昇端
      ANI     X63  ; ﾚｰﾝ6上段(中間)切出し下降端
      OUT     M242  ; ﾚｰﾝ6上段(中間)切出し上昇端
2165  LD      X63  ; ﾚｰﾝ6上段(中間)切出し下降端
      ANI     X62  ; ﾚｰﾝ6上段(中間)切出し上昇端
      OUT     M243  ; ﾚｰﾝ6上段(中間)切出し下降端
2168  LDI     X66  ; ﾚｰﾝ6下段(中間)ﾜｰｸｽﾄｯﾊﾟｰ開端
      OUT     T141 K10  ; ﾚｰﾝ6下段(中間)ﾜｰｸｽﾄｯﾊﾟｰ開端OFF
2173  LD      X65  ; ﾚｰﾝ6下段(中間)ﾜｰｸｽﾄｯﾊﾟｰ閉端
      OR      T141  ; ﾚｰﾝ6下段(中間)ﾜｰｸｽﾄｯﾊﾟｰ開端OFF
      ANI     X66  ; ﾚｰﾝ6下段(中間)ﾜｰｸｽﾄｯﾊﾟｰ開端
      OUT     M244  ; ﾚｰﾝ6下段(中間)ﾜｰｸｽﾄｯﾊﾟｰ閉端
2177  LD      X66  ; ﾚｰﾝ6下段(中間)ﾜｰｸｽﾄｯﾊﾟｰ開端
      ANI     X65  ; ﾚｰﾝ6下段(中間)ﾜｰｸｽﾄｯﾊﾟｰ閉端
      OUT     M245  ; ﾚｰﾝ6下段(中間)ﾜｰｸｽﾄｯﾊﾟｰ開端
2180  LD      X67  ; ﾚｰﾝ6下段(中間)切出し上昇端
      ANI     X68  ; ﾚｰﾝ6下段(中間)切出し下降端
      OUT     M246  ; ﾚｰﾝ6下段(中間)切出し上昇端
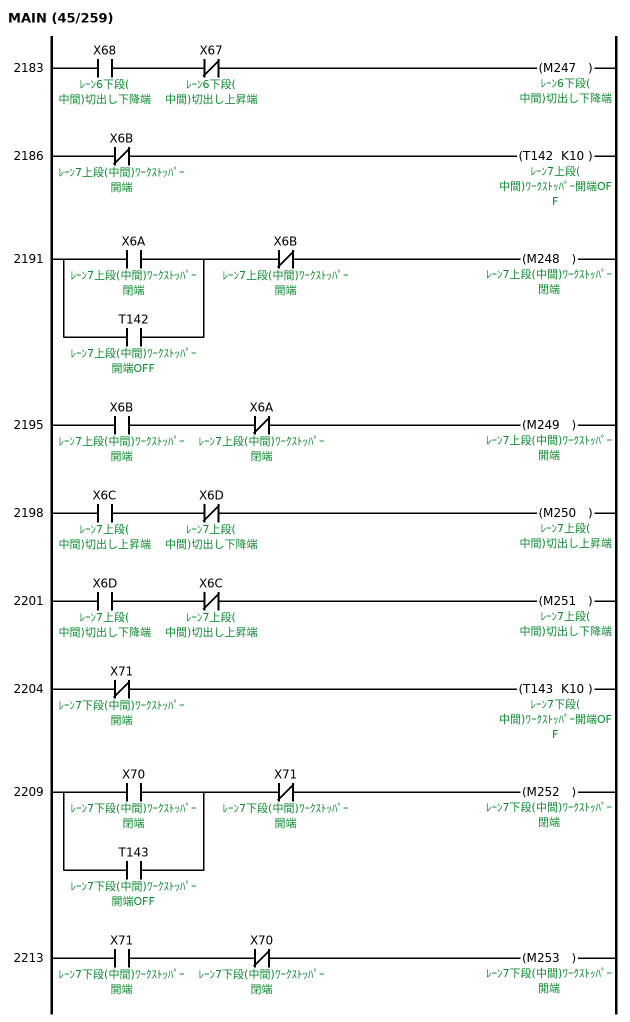
2183  LD      X68  ; ﾚｰﾝ6下段(中間)切出し下降端
      ANI     X67  ; ﾚｰﾝ6下段(中間)切出し上昇端
      OUT     M247  ; ﾚｰﾝ6下段(中間)切出し下降端
2186  LDI     X6B  ; ﾚｰﾝ7上段(中間)ﾜｰｸｽﾄｯﾊﾟｰ開端
      OUT     T142 K10  ; ﾚｰﾝ7上段(中間)ﾜｰｸｽﾄｯﾊﾟｰ開端OFF
2191  LD      X6A  ; ﾚｰﾝ7上段(中間)ﾜｰｸｽﾄｯﾊﾟｰ閉端
      OR      T142  ; ﾚｰﾝ7上段(中間)ﾜｰｸｽﾄｯﾊﾟｰ開端OFF
      ANI     X6B  ; ﾚｰﾝ7上段(中間)ﾜｰｸｽﾄｯﾊﾟｰ開端
      OUT     M248  ; ﾚｰﾝ7上段(中間)ﾜｰｸｽﾄｯﾊﾟｰ閉端
2195  LD      X6B  ; ﾚｰﾝ7上段(中間)ﾜｰｸｽﾄｯﾊﾟｰ開端
      ANI     X6A  ; ﾚｰﾝ7上段(中間)ﾜｰｸｽﾄｯﾊﾟｰ閉端
      OUT     M249  ; ﾚｰﾝ7上段(中間)ﾜｰｸｽﾄｯﾊﾟｰ開端
2198  LD      X6C  ; ﾚｰﾝ7上段(中間)切出し上昇端
      ANI     X6D  ; ﾚｰﾝ7上段(中間)切出し下降端
      OUT     M250  ; ﾚｰﾝ7上段(中間)切出し上昇端
2201  LD      X6D  ; ﾚｰﾝ7上段(中間)切出し下降端
      ANI     X6C  ; ﾚｰﾝ7上段(中間)切出し上昇端
      OUT     M251  ; ﾚｰﾝ7上段(中間)切出し下降端
2204  LDI     X71  ; ﾚｰﾝ7下段(中間)ﾜｰｸｽﾄｯﾊﾟｰ開端
      OUT     T143 K10  ; ﾚｰﾝ7下段(中間)ﾜｰｸｽﾄｯﾊﾟｰ開端OFF
2209  LD      X70  ; ﾚｰﾝ7下段(中間)ﾜｰｸｽﾄｯﾊﾟｰ閉端
      OR      T143  ; ﾚｰﾝ7下段(中間)ﾜｰｸｽﾄｯﾊﾟｰ開端OFF
      ANI     X71  ; ﾚｰﾝ7下段(中間)ﾜｰｸｽﾄｯﾊﾟｰ開端
      OUT     M252  ; ﾚｰﾝ7下段(中間)ﾜｰｸｽﾄｯﾊﾟｰ閉端
2213  LD      X71  ; ﾚｰﾝ7下段(中間)ﾜｰｸｽﾄｯﾊﾟｰ開端
      ANI     X70  ; ﾚｰﾝ7下段(中間)ﾜｰｸｽﾄｯﾊﾟｰ閉端
      OUT     M253  ; ﾚｰﾝ7下段(中間)ﾜｰｸｽﾄｯﾊﾟｰ開端
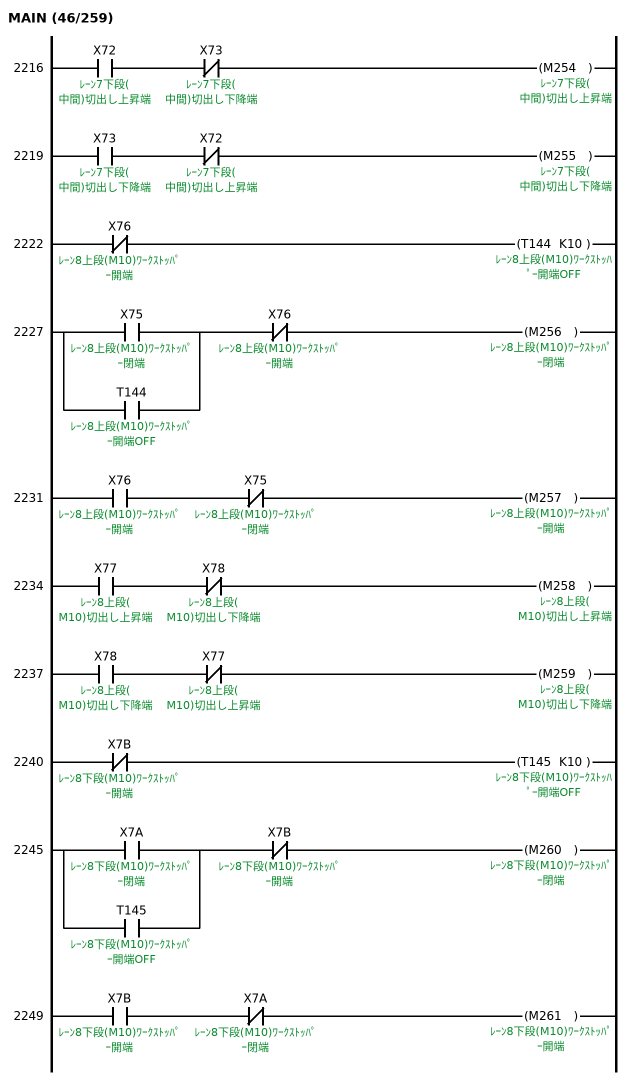
2216  LD      X72  ; ﾚｰﾝ7下段(中間)切出し上昇端
      ANI     X73  ; ﾚｰﾝ7下段(中間)切出し下降端
      OUT     M254  ; ﾚｰﾝ7下段(中間)切出し上昇端
2219  LD      X73  ; ﾚｰﾝ7下段(中間)切出し下降端
      ANI     X72  ; ﾚｰﾝ7下段(中間)切出し上昇端
      OUT     M255  ; ﾚｰﾝ7下段(中間)切出し下降端
2222  LDI     X76  ; ﾚｰﾝ8上段(M10)ﾜｰｸｽﾄｯﾊﾟｰ開端
      OUT     T144 K10  ; ﾚｰﾝ8上段(M10)ﾜｰｸｽﾄｯﾊﾟｰ開端OFF
2227  LD      X75  ; ﾚｰﾝ8上段(M10)ﾜｰｸｽﾄｯﾊﾟｰ閉端
      OR      T144  ; ﾚｰﾝ8上段(M10)ﾜｰｸｽﾄｯﾊﾟｰ開端OFF
      ANI     X76  ; ﾚｰﾝ8上段(M10)ﾜｰｸｽﾄｯﾊﾟｰ開端
      OUT     M256  ; ﾚｰﾝ8上段(M10)ﾜｰｸｽﾄｯﾊﾟｰ閉端
2231  LD      X76  ; ﾚｰﾝ8上段(M10)ﾜｰｸｽﾄｯﾊﾟｰ開端
      ANI     X75  ; ﾚｰﾝ8上段(M10)ﾜｰｸｽﾄｯﾊﾟｰ閉端
      OUT     M257  ; ﾚｰﾝ8上段(M10)ﾜｰｸｽﾄｯﾊﾟｰ開端
2234  LD      X77  ; ﾚｰﾝ8上段(M10)切出し上昇端
      ANI     X78  ; ﾚｰﾝ8上段(M10)切出し下降端
      OUT     M258  ; ﾚｰﾝ8上段(M10)切出し上昇端
2237  LD      X78  ; ﾚｰﾝ8上段(M10)切出し下降端
      ANI     X77  ; ﾚｰﾝ8上段(M10)切出し上昇端
      OUT     M259  ; ﾚｰﾝ8上段(M10)切出し下降端
2240  LDI     X7B  ; ﾚｰﾝ8下段(M10)ﾜｰｸｽﾄｯﾊﾟｰ開端
      OUT     T145 K10  ; ﾚｰﾝ8下段(M10)ﾜｰｸｽﾄｯﾊﾟｰ開端OFF
2245  LD      X7A  ; ﾚｰﾝ8下段(M10)ﾜｰｸｽﾄｯﾊﾟｰ閉端
      OR      T145  ; ﾚｰﾝ8下段(M10)ﾜｰｸｽﾄｯﾊﾟｰ開端OFF
      ANI     X7B  ; ﾚｰﾝ8下段(M10)ﾜｰｸｽﾄｯﾊﾟｰ開端
      OUT     M260  ; ﾚｰﾝ8下段(M10)ﾜｰｸｽﾄｯﾊﾟｰ閉端
2249  LD      X7B  ; ﾚｰﾝ8下段(M10)ﾜｰｸｽﾄｯﾊﾟｰ開端
      ANI     X7A  ; ﾚｰﾝ8下段(M10)ﾜｰｸｽﾄｯﾊﾟｰ閉端
      OUT     M261  ; ﾚｰﾝ8下段(M10)ﾜｰｸｽﾄｯﾊﾟｰ開端
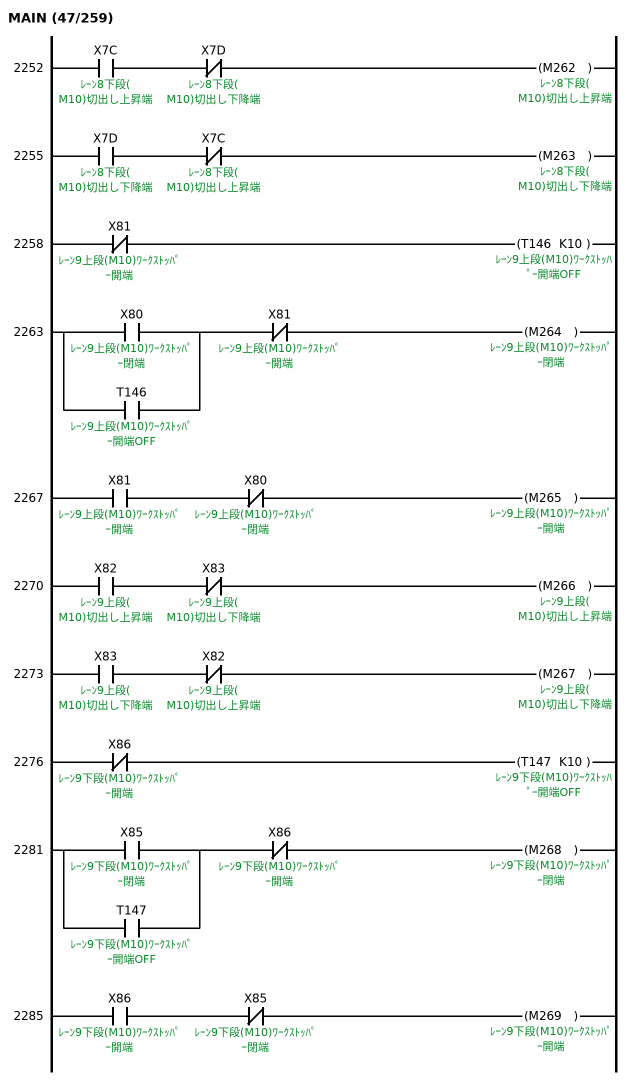
2252  LD      X7C  ; ﾚｰﾝ8下段(M10)切出し上昇端
      ANI     X7D  ; ﾚｰﾝ8下段(M10)切出し下降端
      OUT     M262  ; ﾚｰﾝ8下段(M10)切出し上昇端
2255  LD      X7D  ; ﾚｰﾝ8下段(M10)切出し下降端
      ANI     X7C  ; ﾚｰﾝ8下段(M10)切出し上昇端
      OUT     M263  ; ﾚｰﾝ8下段(M10)切出し下降端
2258  LDI     X81  ; ﾚｰﾝ9上段(M10)ﾜｰｸｽﾄｯﾊﾟｰ開端
      OUT     T146 K10  ; ﾚｰﾝ9上段(M10)ﾜｰｸｽﾄｯﾊﾟｰ開端OFF
2263  LD      X80  ; ﾚｰﾝ9上段(M10)ﾜｰｸｽﾄｯﾊﾟｰ閉端
      OR      T146  ; ﾚｰﾝ9上段(M10)ﾜｰｸｽﾄｯﾊﾟｰ開端OFF
      ANI     X81  ; ﾚｰﾝ9上段(M10)ﾜｰｸｽﾄｯﾊﾟｰ開端
      OUT     M264  ; ﾚｰﾝ9上段(M10)ﾜｰｸｽﾄｯﾊﾟｰ閉端
2267  LD      X81  ; ﾚｰﾝ9上段(M10)ﾜｰｸｽﾄｯﾊﾟｰ開端
      ANI     X80  ; ﾚｰﾝ9上段(M10)ﾜｰｸｽﾄｯﾊﾟｰ閉端
      OUT     M265  ; ﾚｰﾝ9上段(M10)ﾜｰｸｽﾄｯﾊﾟｰ開端
2270  LD      X82  ; ﾚｰﾝ9上段(M10)切出し上昇端
      ANI     X83  ; ﾚｰﾝ9上段(M10)切出し下降端
      OUT     M266  ; ﾚｰﾝ9上段(M10)切出し上昇端
2273  LD      X83  ; ﾚｰﾝ9上段(M10)切出し下降端
      ANI     X82  ; ﾚｰﾝ9上段(M10)切出し上昇端
      OUT     M267  ; ﾚｰﾝ9上段(M10)切出し下降端
2276  LDI     X86  ; ﾚｰﾝ9下段(M10)ﾜｰｸｽﾄｯﾊﾟｰ開端
      OUT     T147 K10  ; ﾚｰﾝ9下段(M10)ﾜｰｸｽﾄｯﾊﾟｰ開端OFF
2281  LD      X85  ; ﾚｰﾝ9下段(M10)ﾜｰｸｽﾄｯﾊﾟｰ閉端
      OR      T147  ; ﾚｰﾝ9下段(M10)ﾜｰｸｽﾄｯﾊﾟｰ開端OFF
      ANI     X86  ; ﾚｰﾝ9下段(M10)ﾜｰｸｽﾄｯﾊﾟｰ開端
      OUT     M268  ; ﾚｰﾝ9下段(M10)ﾜｰｸｽﾄｯﾊﾟｰ閉端
2285  LD      X86  ; ﾚｰﾝ9下段(M10)ﾜｰｸｽﾄｯﾊﾟｰ開端
      ANI     X85  ; ﾚｰﾝ9下段(M10)ﾜｰｸｽﾄｯﾊﾟｰ閉端
      OUT     M269  ; ﾚｰﾝ9下段(M10)ﾜｰｸｽﾄｯﾊﾟｰ開端
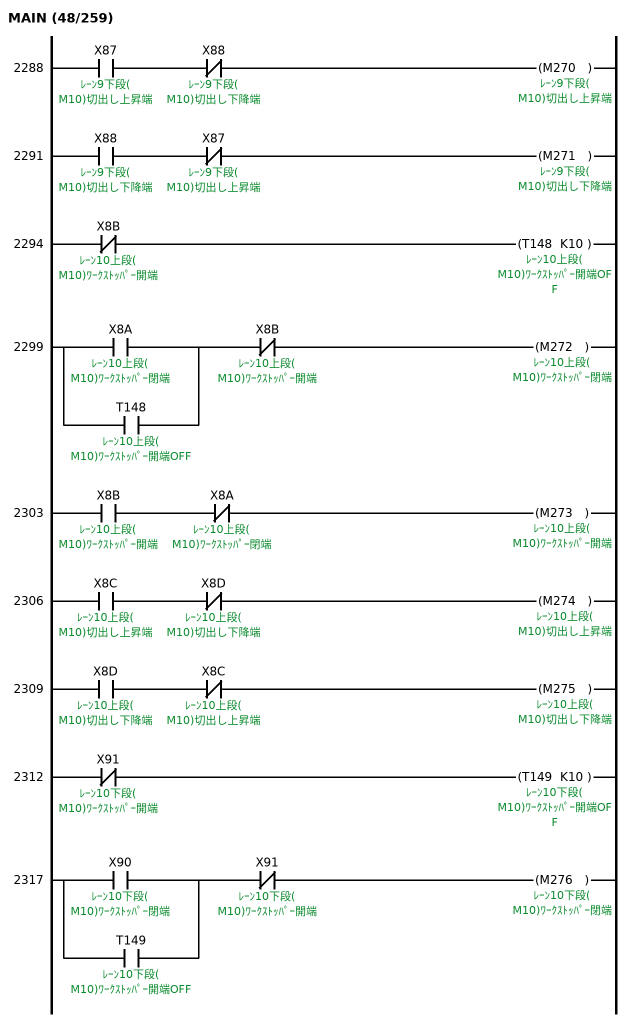
2288  LD      X87  ; ﾚｰﾝ9下段(M10)切出し上昇端
      ANI     X88  ; ﾚｰﾝ9下段(M10)切出し下降端
      OUT     M270  ; ﾚｰﾝ9下段(M10)切出し上昇端
2291  LD      X88  ; ﾚｰﾝ9下段(M10)切出し下降端
      ANI     X87  ; ﾚｰﾝ9下段(M10)切出し上昇端
      OUT     M271  ; ﾚｰﾝ9下段(M10)切出し下降端
2294  LDI     X8B  ; ﾚｰﾝ10上段(M10)ﾜｰｸｽﾄｯﾊﾟｰ開端
      OUT     T148 K10  ; ﾚｰﾝ10上段(M10)ﾜｰｸｽﾄｯﾊﾟｰ開端OFF
2299  LD      X8A  ; ﾚｰﾝ10上段(M10)ﾜｰｸｽﾄｯﾊﾟｰ閉端
      OR      T148  ; ﾚｰﾝ10上段(M10)ﾜｰｸｽﾄｯﾊﾟｰ開端OFF
      ANI     X8B  ; ﾚｰﾝ10上段(M10)ﾜｰｸｽﾄｯﾊﾟｰ開端
      OUT     M272  ; ﾚｰﾝ10上段(M10)ﾜｰｸｽﾄｯﾊﾟｰ閉端
2303  LD      X8B  ; ﾚｰﾝ10上段(M10)ﾜｰｸｽﾄｯﾊﾟｰ開端
      ANI     X8A  ; ﾚｰﾝ10上段(M10)ﾜｰｸｽﾄｯﾊﾟｰ閉端
      OUT     M273  ; ﾚｰﾝ10上段(M10)ﾜｰｸｽﾄｯﾊﾟｰ開端
2306  LD      X8C  ; ﾚｰﾝ10上段(M10)切出し上昇端
      ANI     X8D  ; ﾚｰﾝ10上段(M10)切出し下降端
      OUT     M274  ; ﾚｰﾝ10上段(M10)切出し上昇端
2309  LD      X8D  ; ﾚｰﾝ10上段(M10)切出し下降端
      ANI     X8C  ; ﾚｰﾝ10上段(M10)切出し上昇端
      OUT     M275  ; ﾚｰﾝ10上段(M10)切出し下降端
2312  LDI     X91  ; ﾚｰﾝ10下段(M10)ﾜｰｸｽﾄｯﾊﾟｰ開端
      OUT     T149 K10  ; ﾚｰﾝ10下段(M10)ﾜｰｸｽﾄｯﾊﾟｰ開端OFF
2317  LD      X90  ; ﾚｰﾝ10下段(M10)ﾜｰｸｽﾄｯﾊﾟｰ閉端
      OR      T149  ; ﾚｰﾝ10下段(M10)ﾜｰｸｽﾄｯﾊﾟｰ開端OFF
      ANI     X91  ; ﾚｰﾝ10下段(M10)ﾜｰｸｽﾄｯﾊﾟｰ開端
      OUT     M276  ; ﾚｰﾝ10下段(M10)ﾜｰｸｽﾄｯﾊﾟｰ閉端
